   DATA[1411,38] := 0.000128152;
   DATA[1411,39] := 1.0;
   DATA[1412,1] := 812.7283;
   DATA[1412,2] := 1.0;
   DATA[1412,3] := 1.0;
   DATA[1412,4] := 262.5609;
   DATA[1412,5] := 8.46501;
   DATA[1412,6] := 318.2517;
   DATA[1412,8] := 1.0;
   DATA[1412,9] := 1.0;
   DATA[1412,10] := 1.0;
   DATA[1412,11] := 19.69076;
   DATA[1412,12] := 2.216699;
   DATA[1412,13] := 979.9971;
   DATA[1412,14] := 1.0;
   DATA[1412,15] := 2.0;
   DATA[1412,16] := 1.0;
   DATA[1412,17] := 1.0;
   DATA[1412,18] := 1.0;
   DATA[1412,19] := 2.0;
   DATA[1412,20] := 148.808;
   DATA[1412,21] := 153.5247;
   DATA[1412,22] := 1.7057;
   DATA[1412,23] := 779.3771;
   DATA[1412,24] := 2.0;
   DATA[1412,25] := 2.0;
   DATA[1412,26] := 7.877019;
   DATA[1412,27] := 142.707;
   DATA[1412,28] := 263.1056;
   DATA[1412,29] := 12.11228;
   DATA[1412,30] := 1.718662;
   DATA[1412,31] := 1.271679;
   DATA[1412,32] := 0.7352687;
   DATA[1412,33] := 0.3083624;
   DATA[1412,34] := 2.0;
   DATA[1412,35] := 249.5834;
   DATA[1412,36] := 1.569859;
   DATA[1412,37] := 188.4933;
   DATA[1412,38] := 0.000128152;
   DATA[1412,39] := 1.0;
   DATA[1413,1] := 813.1209;
   DATA[1413,2] := 1.0;
   DATA[1413,3] := 1.0;
   DATA[1413,4] := 262.5609;
   DATA[1413,5] := 8.46501;
   DATA[1413,6] := 318.2517;
   DATA[1413,8] := 1.0;
   DATA[1413,9] := 1.0;
   DATA[1413,10] := 1.0;
   DATA[1413,11] := 19.69076;
   DATA[1413,12] := 2.218621;
   DATA[1413,13] := 979.6367;
   DATA[1413,14] := 1.0;
   DATA[1413,15] := 2.0;
   DATA[1413,16] := 1.0;
   DATA[1413,17] := 1.0;
   DATA[1413,18] := 1.0;
   DATA[1413,19] := 2.0;
   DATA[1413,20] := 148.808;
   DATA[1413,21] := 153.5247;
   DATA[1413,22] := 1.709672;
   DATA[1413,23] := 779.6462;
   DATA[1413,24] := 2.0;
   DATA[1413,25] := 2.0;
   DATA[1413,26] := 7.874776;
   DATA[1413,27] := 142.707;
   DATA[1413,28] := 263.1056;
   DATA[1413,29] := 12.11228;
   DATA[1413,30] := 1.720328;
   DATA[1413,31] := 1.277315;
   DATA[1413,32] := 0.7352687;
   DATA[1413,33] := 0.3083624;
   DATA[1413,34] := 2.0;
   DATA[1413,35] := 249.5834;
   DATA[1413,36] := 1.617916;
   DATA[1413,37] := 188.4933;
   DATA[1413,38] := 0.000128152;
   DATA[1413,39] := 1.0;
   DATA[1414,1] := 812.6498;
   DATA[1414,2] := 1.0;
   DATA[1414,3] := 1.0;
   DATA[1414,4] := 262.5609;
   DATA[1414,5] := 8.46501;
   DATA[1414,6] := 318.2517;
   DATA[1414,8] := 1.0;
   DATA[1414,9] := 1.0;
   DATA[1414,10] := 1.0;
   DATA[1414,11] := 19.69076;
   DATA[1414,12] := 2.218621;
   DATA[1414,13] := 978.9557;
   DATA[1414,14] := 1.0;
   DATA[1414,15] := 2.0;
   DATA[1414,16] := 1.0;
   DATA[1414,17] := 1.0;
   DATA[1414,18] := 1.0;
   DATA[1414,19] := 2.0;
   DATA[1414,20] := 148.808;
   DATA[1414,21] := 153.5247;
   DATA[1414,22] := 1.710057;
   DATA[1414,23] := 779.6847;
   DATA[1414,24] := 2.0;
   DATA[1414,25] := 2.0;
   DATA[1414,26] := 7.874776;
   DATA[1414,27] := 142.707;
   DATA[1414,28] := 263.1056;
   DATA[1414,29] := 12.11228;
   DATA[1414,30] := 1.721097;
   DATA[1414,31] := 1.272064;
   DATA[1414,32] := 0.7352687;
   DATA[1414,33] := 0.3083624;
   DATA[1414,34] := 2.0;
   DATA[1414,35] := 249.5834;
   DATA[1414,36] := 1.617916;
   DATA[1414,37] := 188.4933;
   DATA[1414,38] := 0.000128152;
   DATA[1414,39] := 1.0;
   DATA[1415,1] := 812.5714;
   DATA[1415,2] := 1.0;
   DATA[1415,3] := 1.0;
   DATA[1415,4] := 262.5609;
   DATA[1415,5] := 8.46501;
   DATA[1415,6] := 318.2517;
   DATA[1415,8] := 1.0;
   DATA[1415,9] := 1.0;
   DATA[1415,10] := 1.0;
   DATA[1415,11] := 19.7996;
   DATA[1415,12] := 2.218621;
   DATA[1415,13] := 978.5552;
   DATA[1415,14] := 1.0;
   DATA[1415,15] := 2.0;
   DATA[1415,16] := 1.0;
   DATA[1415,17] := 1.0;
   DATA[1415,18] := 1.0;
   DATA[1415,19] := 2.0;
   DATA[1415,20] := 148.808;
   DATA[1415,21] := 153.5247;
   DATA[1415,22] := 1.710954;
   DATA[1415,23] := 780.0308;
   DATA[1415,24] := 2.0;
   DATA[1415,25] := 2.0;
   DATA[1415,26] := 7.874776;
   DATA[1415,27] := 142.707;
   DATA[1415,28] := 263.1056;
   DATA[1415,29] := 12.11228;
   DATA[1415,30] := 1.722251;
   DATA[1415,31] := 1.271295;
   DATA[1415,32] := 0.7352687;
   DATA[1415,33] := 0.3083624;
   DATA[1415,34] := 2.0;
   DATA[1415,35] := 249.5834;
   DATA[1415,36] := 1.617916;
   DATA[1415,37] := 188.4933;
   DATA[1415,38] := 0.000128152;
   DATA[1415,39] := 1.0;
   DATA[1416,1] := 812.8461;
   DATA[1416,2] := 1.0;
   DATA[1416,3] := 1.0;
   DATA[1416,4] := 262.5609;
   DATA[1416,5] := 8.46501;
   DATA[1416,6] := 318.2517;
   DATA[1416,8] := 1.0;
   DATA[1416,9] := 1.0;
   DATA[1416,10] := 1.0;
   DATA[1416,11] := 19.81881;
   DATA[1416,12] := 2.218621;
   DATA[1416,13] := 978.4351;
   DATA[1416,14] := 1.0;
   DATA[1416,15] := 2.0;
   DATA[1416,16] := 1.0;
   DATA[1416,17] := 1.0;
   DATA[1416,18] := 1.0;
   DATA[1416,19] := 2.0;
   DATA[1416,20] := 148.808;
   DATA[1416,21] := 153.5247;
   DATA[1416,22] := 1.710954;
   DATA[1416,23] := 780.1461;
   DATA[1416,24] := 2.0;
   DATA[1416,25] := 2.0;
   DATA[1416,26] := 7.874776;
   DATA[1416,27] := 142.707;
   DATA[1416,28] := 263.1056;
   DATA[1416,29] := 12.11228;
   DATA[1416,30] := 1.722251;
   DATA[1416,31] := 1.271295;
   DATA[1416,32] := 0.7352687;
   DATA[1416,33] := 0.3083624;
   DATA[1416,34] := 2.0;
   DATA[1416,35] := 249.5834;
   DATA[1416,36] := 1.617916;
   DATA[1416,37] := 188.4933;
   DATA[1416,38] := 0.000128152;
   DATA[1416,39] := 1.0;
   DATA[1417,1] := 812.9246;
   DATA[1417,2] := 1.0;
   DATA[1417,3] := 1.0;
   DATA[1417,4] := 262.5609;
   DATA[1417,5] := 8.46501;
   DATA[1417,6] := 318.2517;
   DATA[1417,8] := 1.0;
   DATA[1417,9] := 1.0;
   DATA[1417,10] := 1.0;
   DATA[1417,11] := 19.81881;
   DATA[1417,12] := 2.218621;
   DATA[1417,13] := 978.0345;
   DATA[1417,14] := 1.0;
   DATA[1417,15] := 2.0;
   DATA[1417,16] := 1.0;
   DATA[1417,17] := 1.0;
   DATA[1417,18] := 1.0;
   DATA[1417,19] := 2.0;
   DATA[1417,20] := 148.808;
   DATA[1417,21] := 153.5247;
   DATA[1417,22] := 1.710954;
   DATA[1417,23] := 780.4537;
   DATA[1417,24] := 2.0;
   DATA[1417,25] := 2.0;
   DATA[1417,26] := 7.874776;
   DATA[1417,27] := 142.707;
   DATA[1417,28] := 263.1056;
   DATA[1417,29] := 12.11228;
   DATA[1417,30] := 1.722251;
   DATA[1417,31] := 1.271295;
   DATA[1417,32] := 0.7352687;
   DATA[1417,33] := 0.3083624;
   DATA[1417,34] := 2.0;
   DATA[1417,35] := 249.5834;
   DATA[1417,36] := 1.617916;
   DATA[1417,37] := 188.4933;
   DATA[1417,38] := 0.000128152;
   DATA[1417,39] := 1.0;
   DATA[1418,1] := 813.0031;
   DATA[1418,2] := 1.0;
   DATA[1418,3] := 1.0;
   DATA[1418,4] := 262.5609;
   DATA[1418,5] := 8.46501;
   DATA[1418,6] := 318.2517;
   DATA[1418,8] := 1.0;
   DATA[1418,9] := 1.0;
   DATA[1418,10] := 1.0;
   DATA[1418,11] := 19.76759;
   DATA[1418,12] := 2.218621;
   DATA[1418,13] := 977.7942;
   DATA[1418,14] := 1.0;
   DATA[1418,15] := 2.0;
   DATA[1418,16] := 1.0;
   DATA[1418,17] := 1.0;
   DATA[1418,18] := 1.0;
   DATA[1418,19] := 2.0;
   DATA[1418,20] := 148.808;
   DATA[1418,21] := 153.5247;
   DATA[1418,22] := 1.710954;
   DATA[1418,23] := 780.7229;
   DATA[1418,24] := 2.0;
   DATA[1418,25] := 2.0;
   DATA[1418,26] := 7.874776;
   DATA[1418,27] := 142.707;
   DATA[1418,28] := 263.1056;
   DATA[1418,29] := 12.11228;
   DATA[1418,30] := 1.722251;
   DATA[1418,31] := 1.262969;
   DATA[1418,32] := 0.7352687;
   DATA[1418,33] := 0.3083624;
   DATA[1418,34] := 2.0;
   DATA[1418,35] := 249.5834;
   DATA[1418,36] := 1.617916;
   DATA[1418,37] := 188.4933;
   DATA[1418,38] := 0.000128152;
   DATA[1418,39] := 1.0;
   DATA[1419,1] := 813.3564;
   DATA[1419,2] := 1.0;
   DATA[1419,3] := 1.0;
   DATA[1419,4] := 262.5609;
   DATA[1419,5] := 8.46501;
   DATA[1419,6] := 318.2517;
   DATA[1419,8] := 1.0;
   DATA[1419,9] := 1.0;
   DATA[1419,10] := 1.0;
   DATA[1419,11] := 19.76759;
   DATA[1419,12] := 2.218621;
   DATA[1419,13] := 977.1533;
   DATA[1419,14] := 1.0;
   DATA[1419,15] := 2.0;
   DATA[1419,16] := 1.0;
   DATA[1419,17] := 1.0;
   DATA[1419,18] := 1.0;
   DATA[1419,19] := 2.0;
   DATA[1419,20] := 148.808;
   DATA[1419,21] := 153.5247;
   DATA[1419,22] := 1.712363;
   DATA[1419,23] := 781.1459;
   DATA[1419,24] := 2.0;
   DATA[1419,25] := 2.0;
   DATA[1419,26] := 7.87766;
   DATA[1419,27] := 142.707;
   DATA[1419,28] := 263.1056;
   DATA[1419,29] := 12.11228;
   DATA[1419,30] := 1.722251;
   DATA[1419,31] := 1.274881;
   DATA[1419,32] := 0.7352687;
   DATA[1419,33] := 0.3083624;
   DATA[1419,34] := 2.0;
   DATA[1419,35] := 249.5834;
   DATA[1419,36] := 1.617916;
   DATA[1419,37] := 188.4933;
   DATA[1419,38] := 0.000128152;
   DATA[1419,39] := 1.0;
   DATA[1420,1] := 813.5527;
   DATA[1420,2] := 1.0;
   DATA[1420,3] := 1.0;
   DATA[1420,4] := 262.5609;
   DATA[1420,5] := 8.46501;
   DATA[1420,6] := 318.3799;
   DATA[1420,8] := 1.0;
   DATA[1420,9] := 1.0;
   DATA[1420,10] := 1.0;
   DATA[1420,11] := 19.73558;
   DATA[1420,12] := 2.218621;
   DATA[1420,13] := 976.5926;
   DATA[1420,14] := 1.0;
   DATA[1420,15] := 2.0;
   DATA[1420,16] := 1.0;
   DATA[1420,17] := 1.0;
   DATA[1420,18] := 1.0;
   DATA[1420,19] := 2.0;
   DATA[1420,20] := 148.808;
   DATA[1420,21] := 153.5247;
   DATA[1420,22] := 1.712363;
   DATA[1420,23] := 780.9536;
   DATA[1420,24] := 2.0;
   DATA[1420,25] := 2.0;
   DATA[1420,26] := 7.87766;
   DATA[1420,27] := 142.707;
   DATA[1420,28] := 263.1056;
   DATA[1420,29] := 12.11228;
   DATA[1420,30] := 1.722251;
   DATA[1420,31] := 1.288203;
   DATA[1420,32] := 0.7352687;
   DATA[1420,33] := 0.3083624;
   DATA[1420,34] := 2.0;
   DATA[1420,35] := 249.5834;
   DATA[1420,36] := 1.617916;
   DATA[1420,37] := 188.4933;
   DATA[1420,38] := 0.000128152;
   DATA[1420,39] := 1.0;
   DATA[1421,1] := 813.7097;
   DATA[1421,2] := 1.0;
   DATA[1421,3] := 1.0;
   DATA[1421,4] := 262.5609;
   DATA[1421,5] := 8.46501;
   DATA[1421,6] := 318.3799;
   DATA[1421,8] := 1.0;
   DATA[1421,9] := 1.0;
   DATA[1421,10] := 1.0;
   DATA[1421,11] := 19.7804;
   DATA[1421,12] := 2.218621;
   DATA[1421,13] := 976.192;
   DATA[1421,14] := 1.0;
   DATA[1421,15] := 2.0;
   DATA[1421,16] := 1.0;
   DATA[1421,17] := 1.0;
   DATA[1421,18] := 1.0;
   DATA[1421,19] := 2.0;
   DATA[1421,20] := 148.808;
   DATA[1421,21] := 153.5247;
   DATA[1421,22] := 1.712363;
   DATA[1421,23] := 781.2228;
   DATA[1421,24] := 2.0;
   DATA[1421,25] := 2.0;
   DATA[1421,26] := 7.87766;
   DATA[1421,27] := 142.707;
   DATA[1421,28] := 263.1056;
   DATA[1421,29] := 12.11228;
   DATA[1421,30] := 1.722251;
   DATA[1421,31] := 1.29781;
   DATA[1421,32] := 0.7352687;
   DATA[1421,33] := 0.3083624;
   DATA[1421,34] := 2.0;
   DATA[1421,35] := 249.7597;
   DATA[1421,36] := 1.617916;
   DATA[1421,37] := 188.7016;
   DATA[1421,38] := 0.000128152;
   DATA[1421,39] := 1.0;
   DATA[1422,1] := 813.5134;
   DATA[1422,2] := 1.0;
   DATA[1422,3] := 1.0;
   DATA[1422,4] := 262.5609;
   DATA[1422,5] := 8.46501;
   DATA[1422,6] := 318.3799;
   DATA[1422,8] := 1.0;
   DATA[1422,9] := 1.0;
   DATA[1422,10] := 1.0;
   DATA[1422,11] := 19.7804;
   DATA[1422,12] := 2.218621;
   DATA[1422,13] := 975.5511;
   DATA[1422,14] := 1.0;
   DATA[1422,15] := 2.0;
   DATA[1422,16] := 1.0;
   DATA[1422,17] := 1.0;
   DATA[1422,18] := 1.0;
   DATA[1422,19] := 2.0;
   DATA[1422,20] := 148.808;
   DATA[1422,21] := 153.5247;
   DATA[1422,22] := 1.710698;
   DATA[1422,23] := 781.415;
   DATA[1422,24] := 2.0;
   DATA[1422,25] := 2.0;
   DATA[1422,26] := 7.87766;
   DATA[1422,27] := 142.707;
   DATA[1422,28] := 263.1056;
   DATA[1422,29] := 12.11228;
   DATA[1422,30] := 1.722251;
   DATA[1422,31] := 1.30921;
   DATA[1422,32] := 0.7352687;
   DATA[1422,33] := 0.3083624;
   DATA[1422,34] := 2.0;
   DATA[1422,35] := 249.8398;
   DATA[1422,36] := 1.617916;
   DATA[1422,37] := 188.7657;
   DATA[1422,38] := 0.000128152;
   DATA[1422,39] := 1.0;
   DATA[1423,1] := 813.6312;
   DATA[1423,2] := 1.0;
   DATA[1423,3] := 1.0;
   DATA[1423,4] := 262.5609;
   DATA[1423,5] := 8.46501;
   DATA[1423,6] := 318.3799;
   DATA[1423,8] := 1.0;
   DATA[1423,9] := 1.0;
   DATA[1423,10] := 1.0;
   DATA[1423,11] := 19.7804;
   DATA[1423,12] := 2.216699;
   DATA[1423,13] := 975.0305;
   DATA[1423,14] := 1.0;
   DATA[1423,15] := 2.0;
   DATA[1423,16] := 1.0;
   DATA[1423,17] := 1.0;
   DATA[1423,18] := 1.0;
   DATA[1423,19] := 2.0;
   DATA[1423,20] := 148.808;
   DATA[1423,21] := 153.5247;
   DATA[1423,22] := 1.7098;
   DATA[1423,23] := 781.3381;
   DATA[1423,24] := 2.0;
   DATA[1423,25] := 2.0;
   DATA[1423,26] := 7.87766;
   DATA[1423,27] := 142.707;
   DATA[1423,28] := 263.1056;
   DATA[1423,29] := 12.11228;
   DATA[1423,30] := 1.722251;
   DATA[1423,31] := 1.311643;
   DATA[1423,32] := 0.7359089;
   DATA[1423,33] := 0.3083624;
   DATA[1423,34] := 2.0;
   DATA[1423,35] := 249.8398;
   DATA[1423,36] := 1.617916;
   DATA[1423,37] := 188.7657;
   DATA[1423,38] := 0.000128152;
   DATA[1423,39] := 1.0;
   DATA[1424,1] := 813.7097;
   DATA[1424,2] := 1.0;
   DATA[1424,3] := 1.0;
   DATA[1424,4] := 262.5609;
   DATA[1424,5] := 8.46501;
   DATA[1424,6] := 318.3799;
   DATA[1424,8] := 1.0;
   DATA[1424,9] := 1.0;
   DATA[1424,10] := 1.0;
   DATA[1424,11] := 19.67796;
   DATA[1424,12] := 2.216699;
   DATA[1424,13] := 974.7902;
   DATA[1424,14] := 1.0;
   DATA[1424,15] := 2.0;
   DATA[1424,16] := 1.0;
   DATA[1424,17] := 1.0;
   DATA[1424,18] := 1.0;
   DATA[1424,19] := 2.0;
   DATA[1424,20] := 148.808;
   DATA[1424,21] := 153.5247;
   DATA[1424,22] := 1.7098;
   DATA[1424,23] := 781.5304;
   DATA[1424,24] := 2.0;
   DATA[1424,25] := 2.0;
   DATA[1424,26] := 7.87766;
   DATA[1424,27] := 142.707;
   DATA[1424,28] := 263.1056;
   DATA[1424,29] := 12.11228;
   DATA[1424,30] := 1.720841;
   DATA[1424,31] := 1.302037;
   DATA[1424,32] := 0.736549;
   DATA[1424,33] := 0.3083624;
   DATA[1424,34] := 2.0;
   DATA[1424,35] := 249.8398;
   DATA[1424,36] := 1.617916;
   DATA[1424,37] := 188.7657;
   DATA[1424,38] := 0.000128152;
   DATA[1424,39] := 1.0;
   DATA[1425,1] := 813.6312;
   DATA[1425,2] := 1.0;
   DATA[1425,3] := 1.0;
   DATA[1425,4] := 262.5609;
   DATA[1425,5] := 8.46501;
   DATA[1425,6] := 318.3799;
   DATA[1425,8] := 1.0;
   DATA[1425,9] := 1.0;
   DATA[1425,10] := 1.0;
   DATA[1425,11] := 19.67796;
   DATA[1425,12] := 2.218621;
   DATA[1425,13] := 974.6299;
   DATA[1425,14] := 1.0;
   DATA[1425,15] := 2.0;
   DATA[1425,16] := 1.0;
   DATA[1425,17] := 1.0;
   DATA[1425,18] := 1.0;
   DATA[1425,19] := 2.0;
   DATA[1425,20] := 148.808;
   DATA[1425,21] := 153.5247;
   DATA[1425,22] := 1.7098;
   DATA[1425,23] := 781.6073;
   DATA[1425,24] := 2.0;
   DATA[1425,25] := 2.0;
   DATA[1425,26] := 7.87766;
   DATA[1425,27] := 142.707;
   DATA[1425,28] := 263.1056;
   DATA[1425,29] := 12.11228;
   DATA[1425,30] := 1.718662;
   DATA[1425,31] := 1.302037;
   DATA[1425,32] := 0.736549;
   DATA[1425,33] := 0.3083624;
   DATA[1425,34] := 2.0;
   DATA[1425,35] := 249.8398;
   DATA[1425,36] := 1.617916;
   DATA[1425,37] := 188.7657;
   DATA[1425,38] := 0.000128152;
   DATA[1425,39] := 1.0;
   DATA[1426,1] := 813.1994;
   DATA[1426,2] := 1.0;
   DATA[1426,3] := 1.0;
   DATA[1426,4] := 262.5609;
   DATA[1426,5] := 8.46501;
   DATA[1426,6] := 318.3799;
   DATA[1426,8] := 1.0;
   DATA[1426,9] := 1.0;
   DATA[1426,10] := 1.0;
   DATA[1426,11] := 19.73558;
   DATA[1426,12] := 2.219005;
   DATA[1426,13] := 974.4697;
   DATA[1426,14] := 1.0;
   DATA[1426,15] := 2.0;
   DATA[1426,16] := 1.0;
   DATA[1426,17] := 1.0;
   DATA[1426,18] := 1.0;
   DATA[1426,19] := 2.0;
   DATA[1426,20] := 148.808;
   DATA[1426,21] := 153.5247;
   DATA[1426,22] := 1.7098;
   DATA[1426,23] := 781.9918;
   DATA[1426,24] := 2.0;
   DATA[1426,25] := 2.0;
   DATA[1426,26] := 7.87766;
   DATA[1426,27] := 142.707;
   DATA[1426,28] := 263.1056;
   DATA[1426,29] := 12.11228;
   DATA[1426,30] := 1.718662;
   DATA[1426,31] := 1.295248;
   DATA[1426,32] := 0.7380853;
   DATA[1426,33] := 0.3083624;
   DATA[1426,34] := 2.0;
   DATA[1426,35] := 249.8398;
   DATA[1426,36] := 1.617916;
   DATA[1426,37] := 188.7657;
   DATA[1426,38] := 0.000128152;
   DATA[1426,39] := 1.0;
   DATA[1427,1] := 813.1994;
   DATA[1427,2] := 1.0;
   DATA[1427,3] := 1.0;
   DATA[1427,4] := 262.5609;
   DATA[1427,5] := 8.46501;
   DATA[1427,6] := 318.3799;
   DATA[1427,8] := 1.0;
   DATA[1427,9] := 1.0;
   DATA[1427,10] := 1.0;
   DATA[1427,11] := 19.79;
   DATA[1427,12] := 2.219005;
   DATA[1427,13] := 973.9891;
   DATA[1427,14] := 1.0;
   DATA[1427,15] := 2.0;
   DATA[1427,16] := 1.0;
   DATA[1427,17] := 1.0;
   DATA[1427,18] := 1.0;
   DATA[1427,19] := 2.0;
   DATA[1427,20] := 148.808;
   DATA[1427,21] := 153.5247;
   DATA[1427,22] := 1.7098;
   DATA[1427,23] := 781.7227;
   DATA[1427,24] := 2.0;
   DATA[1427,25] := 2.0;
   DATA[1427,26] := 7.87766;
   DATA[1427,27] := 142.707;
   DATA[1427,28] := 263.1056;
   DATA[1427,29] := 12.11228;
   DATA[1427,30] := 1.718662;
   DATA[1427,31] := 1.282439;
   DATA[1427,32] := 0.7387255;
   DATA[1427,33] := 0.3083624;
   DATA[1427,34] := 2.0;
   DATA[1427,35] := 249.8398;
   DATA[1427,36] := 1.617916;
   DATA[1427,37] := 188.6375;
   DATA[1427,38] := 0.000128152;
   DATA[1427,39] := 1.0;
   DATA[1428,1] := 813.4349;
   DATA[1428,2] := 1.0;
   DATA[1428,3] := 1.0;
   DATA[1428,4] := 262.5609;
   DATA[1428,5] := 8.46501;
   DATA[1428,6] := 318.3799;
   DATA[1428,8] := 1.0;
   DATA[1428,9] := 1.0;
   DATA[1428,10] := 1.0;
   DATA[1428,11] := 19.79;
   DATA[1428,12] := 2.217211;
   DATA[1428,13] := 973.1479;
   DATA[1428,14] := 1.0;
   DATA[1428,15] := 2.0;
   DATA[1428,16] := 1.0;
   DATA[1428,17] := 1.0;
   DATA[1428,18] := 1.0;
   DATA[1428,19] := 2.0;
   DATA[1428,20] := 148.808;
   DATA[1428,21] := 153.5247;
   DATA[1428,22] := 1.7098;
   DATA[1428,23] := 781.8765;
   DATA[1428,24] := 2.0;
   DATA[1428,25] := 2.0;
   DATA[1428,26] := 7.877339;
   DATA[1428,27] := 142.707;
   DATA[1428,28] := 263.1056;
   DATA[1428,29] := 12.11228;
   DATA[1428,30] := 1.718662;
   DATA[1428,31] := 1.272576;
   DATA[1428,32] := 0.7387255;
   DATA[1428,33] := 0.3083624;
   DATA[1428,34] := 2.0;
   DATA[1428,35] := 249.8398;
   DATA[1428,36] := 1.617916;
   DATA[1428,37] := 188.6215;
   DATA[1428,38] := 0.000128152;
   DATA[1428,39] := 1.0;
   DATA[1429,1] := 813.5527;
   DATA[1429,2] := 1.0;
   DATA[1429,3] := 1.0;
   DATA[1429,4] := 262.5609;
   DATA[1429,5] := 8.466932;
   DATA[1429,6] := 318.3799;
   DATA[1429,8] := 1.0;
   DATA[1429,9] := 1.0;
   DATA[1429,10] := 1.0;
   DATA[1429,11] := 19.7804;
   DATA[1429,12] := 2.217211;
   DATA[1429,13] := 972.3869;
   DATA[1429,14] := 1.0;
   DATA[1429,15] := 2.0;
   DATA[1429,16] := 1.0;
   DATA[1429,17] := 1.0;
   DATA[1429,18] := 1.0;
   DATA[1429,19] := 2.0;
   DATA[1429,20] := 148.808;
   DATA[1429,21] := 153.5247;
   DATA[1429,22] := 1.7098;
   DATA[1429,23] := 782.261;
   DATA[1429,24] := 2.0;
   DATA[1429,25] := 2.0;
   DATA[1429,26] := 7.877339;
   DATA[1429,27] := 142.707;
   DATA[1429,28] := 263.1056;
   DATA[1429,29] := 12.11228;
   DATA[1429,30] := 1.718662;
   DATA[1429,31] := 1.262073;
   DATA[1429,32] := 0.7387255;
   DATA[1429,33] := 0.3083624;
   DATA[1429,34] := 2.0;
   DATA[1429,35] := 249.6635;
   DATA[1429,36] := 1.617916;
   DATA[1429,37] := 188.6215;
   DATA[1429,38] := 0.000128152;
   DATA[1429,39] := 1.0;
   DATA[1430,1] := 813.5919;
   DATA[1430,2] := 1.0;
   DATA[1430,3] := 1.0;
   DATA[1430,4] := 262.5609;
   DATA[1430,5] := 8.468855;
   DATA[1430,6] := 318.3799;
   DATA[1430,8] := 1.0;
   DATA[1430,9] := 1.0;
   DATA[1430,10] := 1.0;
   DATA[1430,11] := 19.7804;
   DATA[1430,12] := 2.216827;
   DATA[1430,13] := 972.1466;
   DATA[1430,14] := 1.0;
   DATA[1430,15] := 2.0;
   DATA[1430,16] := 1.0;
   DATA[1430,17] := 1.0;
   DATA[1430,18] := 1.0;
   DATA[1430,19] := 2.0;
   DATA[1430,20] := 148.808;
   DATA[1430,21] := 153.5247;
   DATA[1430,22] := 1.7098;
   DATA[1430,23] := 782.2994;
   DATA[1430,24] := 2.0;
   DATA[1430,25] := 2.0;
   DATA[1430,26] := 7.877339;
   DATA[1430,27] := 142.707;
   DATA[1430,28] := 263.1056;
   DATA[1430,29] := 12.11228;
   DATA[1430,30] := 1.718662;
   DATA[1430,31] := 1.262073;
   DATA[1430,32] := 0.7370611;
   DATA[1430,33] := 0.3083624;
   DATA[1430,34] := 2.0;
   DATA[1430,35] := 249.6635;
   DATA[1430,36] := 1.617916;
   DATA[1430,37] := 188.6215;
   DATA[1430,38] := 0.000128152;
   DATA[1430,39] := 1.0;
   DATA[1431,1] := 813.7489;
   DATA[1431,2] := 1.0;
   DATA[1431,3] := 1.0;
   DATA[1431,4] := 262.5609;
   DATA[1431,5] := 8.468855;
   DATA[1431,6] := 318.3799;
   DATA[1431,8] := 1.0;
   DATA[1431,9] := 1.0;
   DATA[1431,10] := 1.0;
   DATA[1431,11] := 19.7804;
   DATA[1431,12] := 2.216827;
   DATA[1431,13] := 971.5858;
   DATA[1431,14] := 1.0;
   DATA[1431,15] := 2.0;
   DATA[1431,16] := 1.0;
   DATA[1431,17] := 1.0;
   DATA[1431,18] := 1.0;
   DATA[1431,19] := 2.0;
   DATA[1431,20] := 148.808;
   DATA[1431,21] := 153.5247;
   DATA[1431,22] := 1.711466;
   DATA[1431,23] := 782.2994;
   DATA[1431,24] := 2.0;
   DATA[1431,25] := 2.0;
   DATA[1431,26] := 7.876058;
   DATA[1431,27] := 142.707;
   DATA[1431,28] := 263.1056;
   DATA[1431,29] := 12.11228;
   DATA[1431,30] := 1.719046;
   DATA[1431,31] := 1.280646;
   DATA[1431,32] := 0.7355248;
   DATA[1431,33] := 0.3083624;
   DATA[1431,34] := 2.0;
   DATA[1431,35] := 249.6635;
   DATA[1431,36] := 1.617916;
   DATA[1431,37] := 188.6215;
   DATA[1431,38] := 0.000128152;
   DATA[1431,39] := 1.0;
   DATA[1432,1] := 813.6312;
   DATA[1432,2] := 1.0;
   DATA[1432,3] := 1.0;
   DATA[1432,4] := 262.5609;
   DATA[1432,5] := 8.468855;
   DATA[1432,6] := 318.3799;
   DATA[1432,8] := 1.0;
   DATA[1432,9] := 1.0;
   DATA[1432,10] := 1.0;
   DATA[1432,11] := 19.7804;
   DATA[1432,12] := 2.216827;
   DATA[1432,13] := 971.2253;
   DATA[1432,14] := 1.0;
   DATA[1432,15] := 2.0;
   DATA[1432,16] := 1.0;
   DATA[1432,17] := 1.0;
   DATA[1432,18] := 1.0;
   DATA[1432,19] := 2.0;
   DATA[1432,20] := 148.808;
   DATA[1432,21] := 153.5247;
   DATA[1432,22] := 1.711466;
   DATA[1432,23] := 782.261;
   DATA[1432,24] := 2.0;
   DATA[1432,25] := 2.0;
   DATA[1432,26] := 7.875737;
   DATA[1432,27] := 142.707;
   DATA[1432,28] := 263.1056;
   DATA[1432,29] := 12.11228;
   DATA[1432,30] := 1.719559;
   DATA[1432,31] := 1.292558;
   DATA[1432,32] := 0.7352687;
   DATA[1432,33] := 0.3083624;
   DATA[1432,34] := 2.0;
   DATA[1432,35] := 249.6635;
   DATA[1432,36] := 1.617916;
   DATA[1432,37] := 188.6215;
   DATA[1432,38] := 0.000128152;
   DATA[1432,39] := 1.0;
   DATA[1433,1] := 813.9452;
   DATA[1433,2] := 1.0;
   DATA[1433,3] := 1.0;
   DATA[1433,4] := 262.5609;
   DATA[1433,5] := 8.468855;
   DATA[1433,6] := 318.3799;
   DATA[1433,8] := 1.0;
   DATA[1433,9] := 1.0;
   DATA[1433,10] := 1.0;
   DATA[1433,11] := 19.76439;
   DATA[1433,12] := 2.218621;
   DATA[1433,13] := 971.0651;
   DATA[1433,14] := 1.0;
   DATA[1433,15] := 2.0;
   DATA[1433,16] := 1.0;
   DATA[1433,17] := 1.0;
   DATA[1433,18] := 1.0;
   DATA[1433,19] := 2.0;
   DATA[1433,20] := 148.808;
   DATA[1433,21] := 153.5247;
   DATA[1433,22] := 1.711466;
   DATA[1433,23] := 782.4532;
   DATA[1433,24] := 2.0;
   DATA[1433,25] := 2.0;
   DATA[1433,26] := 7.875737;
   DATA[1433,27] := 142.707;
   DATA[1433,28] := 263.1056;
   DATA[1433,29] := 12.11228;
   DATA[1433,30] := 1.72161;
   DATA[1433,31] := 1.292558;
   DATA[1433,32] := 0.7352687;
   DATA[1433,33] := 0.3083624;
   DATA[1433,34] := 2.0;
   DATA[1433,35] := 249.6635;
   DATA[1433,36] := 1.617916;
   DATA[1433,37] := 188.6215;
   DATA[1433,38] := 0.000128152;
   DATA[1433,39] := 1.0;
   DATA[1434,1] := 813.7882;
   DATA[1434,2] := 1.0;
   DATA[1434,3] := 1.0;
   DATA[1434,4] := 262.5609;
   DATA[1434,5] := 8.468855;
   DATA[1434,6] := 318.3799;
   DATA[1434,8] := 1.0;
   DATA[1434,9] := 1.0;
   DATA[1434,10] := 1.0;
   DATA[1434,11] := 19.76439;
   DATA[1434,12] := 2.218621;
   DATA[1434,13] := 970.6245;
   DATA[1434,14] := 1.0;
   DATA[1434,15] := 2.0;
   DATA[1434,16] := 1.0;
   DATA[1434,17] := 1.0;
   DATA[1434,18] := 1.0;
   DATA[1434,19] := 2.0;
   DATA[1434,20] := 148.808;
   DATA[1434,21] := 153.5247;
   DATA[1434,22] := 1.711466;
   DATA[1434,23] := 782.4532;
   DATA[1434,24] := 2.0;
   DATA[1434,25] := 2.0;
   DATA[1434,26] := 7.875737;
   DATA[1434,27] := 142.707;
   DATA[1434,28] := 263.1056;
   DATA[1434,29] := 12.11228;
   DATA[1434,30] := 1.722379;
   DATA[1434,31] := 1.289996;
   DATA[1434,32] := 0.7352687;
   DATA[1434,33] := 0.3083624;
   DATA[1434,34] := 2.0;
   DATA[1434,35] := 249.8558;
   DATA[1434,36] := 1.617916;
   DATA[1434,37] := 188.6215;
   DATA[1434,38] := 0.000128152;
   DATA[1434,39] := 1.0;
   DATA[1435,1] := 813.5134;
   DATA[1435,2] := 1.0;
   DATA[1435,3] := 1.0;
   DATA[1435,4] := 262.5609;
   DATA[1435,5] := 8.466612;
   DATA[1435,6] := 318.3799;
   DATA[1435,8] := 1.0;
   DATA[1435,9] := 1.0;
   DATA[1435,10] := 1.0;
   DATA[1435,11] := 19.84442;
   DATA[1435,12] := 2.217468;
   DATA[1435,13] := 970.264;
   DATA[1435,14] := 1.0;
   DATA[1435,15] := 2.0;
   DATA[1435,16] := 1.0;
   DATA[1435,17] := 1.0;
   DATA[1435,18] := 1.0;
   DATA[1435,19] := 2.0;
   DATA[1435,20] := 148.808;
   DATA[1435,21] := 153.5247;
   DATA[1435,22] := 1.711466;
   DATA[1435,23] := 782.607;
   DATA[1435,24] := 2.0;
   DATA[1435,25] := 2.0;
   DATA[1435,26] := 7.875737;
   DATA[1435,27] := 142.707;
   DATA[1435,28] := 263.0095;
   DATA[1435,29] := 12.11228;
   DATA[1435,30] := 1.722379;
   DATA[1435,31] := 1.281927;
   DATA[1435,32] := 0.7352687;
   DATA[1435,33] := 0.3083624;
   DATA[1435,34] := 2.0;
   DATA[1435,35] := 250.0;
   DATA[1435,36] := 1.617916;
   DATA[1435,37] := 188.8779;
   DATA[1435,38] := 0.000128152;
   DATA[1435,39] := 1.0;
   DATA[1436,1] := 813.3171;
   DATA[1436,2] := 1.0;
   DATA[1436,3] := 1.0;
   DATA[1436,4] := 262.5609;
   DATA[1436,5] := 8.464369;
   DATA[1436,6] := 318.3799;
   DATA[1436,8] := 1.0;
   DATA[1436,9] := 1.0;
   DATA[1436,10] := 1.0;
   DATA[1436,11] := 19.88604;
   DATA[1436,12] := 2.216571;
   DATA[1436,13] := 970.0237;
   DATA[1436,14] := 1.0;
   DATA[1436,15] := 2.0;
   DATA[1436,16] := 1.0;
   DATA[1436,17] := 1.0;
   DATA[1436,18] := 1.0;
   DATA[1436,19] := 2.0;
   DATA[1436,20] := 148.808;
   DATA[1436,21] := 153.5247;
   DATA[1436,22] := 1.711466;
   DATA[1436,23] := 782.7608;
   DATA[1436,24] := 2.0;
   DATA[1436,25] := 2.0;
   DATA[1436,26] := 7.875737;
   DATA[1436,27] := 142.707;
   DATA[1436,28] := 263.0095;
   DATA[1436,29] := 12.11228;
   DATA[1436,30] := 1.722379;
   DATA[1436,31] := 1.281542;
   DATA[1436,32] := 0.7352687;
   DATA[1436,33] := 0.3083624;
   DATA[1436,34] := 2.0;
   DATA[1436,35] := 250.0961;
   DATA[1436,36] := 1.617916;
   DATA[1436,37] := 188.974;
   DATA[1436,38] := 0.000128152;
   DATA[1436,39] := 1.0;
   DATA[1437,1] := 813.1994;
   DATA[1437,2] := 1.0;
   DATA[1437,3] := 1.0;
   DATA[1437,4] := 262.5609;
   DATA[1437,5] := 8.464369;
   DATA[1437,6] := 318.3799;
   DATA[1437,8] := 1.0;
   DATA[1437,9] := 1.0;
   DATA[1437,10] := 1.0;
   DATA[1437,11] := 19.88604;
   DATA[1437,12] := 2.217211;
   DATA[1437,13] := 969.3829;
   DATA[1437,14] := 1.0;
   DATA[1437,15] := 2.0;
   DATA[1437,16] := 1.0;
   DATA[1437,17] := 1.0;
   DATA[1437,18] := 1.0;
   DATA[1437,19] := 2.0;
   DATA[1437,20] := 148.808;
   DATA[1437,21] := 153.5247;
   DATA[1437,22] := 1.711466;
   DATA[1437,23] := 782.9531;
   DATA[1437,24] := 2.0;
   DATA[1437,25] := 2.0;
   DATA[1437,26] := 7.875737;
   DATA[1437,27] := 142.707;
   DATA[1437,28] := 263.0095;
   DATA[1437,29] := 12.11228;
   DATA[1437,30] := 1.72443;
   DATA[1437,31] := 1.282439;
   DATA[1437,32] := 0.7352687;
   DATA[1437,33] := 0.3083624;
   DATA[1437,34] := 2.0;
   DATA[1437,35] := 250.2243;
   DATA[1437,36] := 1.649953;
   DATA[1437,37] := 188.974;
   DATA[1437,38] := 0.000128152;
   DATA[1437,39] := 1.0;
   DATA[1438,1] := 813.2386;
   DATA[1438,2] := 1.0;
   DATA[1438,3] := 1.0;
   DATA[1438,4] := 262.5609;
   DATA[1438,5] := 8.464369;
   DATA[1438,6] := 318.3799;
   DATA[1438,8] := 1.0;
   DATA[1438,9] := 1.0;
   DATA[1438,10] := 1.0;
   DATA[1438,11] := 19.7996;
   DATA[1438,12] := 2.217211;
   DATA[1438,13] := 968.8622;
   DATA[1438,14] := 1.0;
   DATA[1438,15] := 2.0;
   DATA[1438,16] := 1.0;
   DATA[1438,17] := 1.0;
   DATA[1438,18] := 1.0;
   DATA[1438,19] := 2.0;
   DATA[1438,20] := 148.808;
   DATA[1438,21] := 153.5247;
   DATA[1438,22] := 1.711466;
   DATA[1438,23] := 783.03;
   DATA[1438,24] := 2.0;
   DATA[1438,25] := 2.0;
   DATA[1438,26] := 7.875737;
   DATA[1438,27] := 142.707;
   DATA[1438,28] := 263.0095;
   DATA[1438,29] := 12.11228;
   DATA[1438,30] := 1.725968;
   DATA[1438,31] := 1.300115;
   DATA[1438,32] := 0.7352687;
   DATA[1438,33] := 0.3083624;
   DATA[1438,34] := 2.0;
   DATA[1438,35] := 250.2243;
   DATA[1438,36] := 1.649953;
   DATA[1438,37] := 189.1022;
   DATA[1438,38] := 0.000128152;
   DATA[1438,39] := 1.0;
   DATA[1439,1] := 813.0424;
   DATA[1439,2] := 1.0;
   DATA[1439,3] := 1.0;
   DATA[1439,4] := 262.5609;
   DATA[1439,5] := 8.464369;
   DATA[1439,6] := 318.3799;
   DATA[1439,8] := 1.0;
   DATA[1439,9] := 1.0;
   DATA[1439,10] := 1.0;
   DATA[1439,11] := 19.73558;
   DATA[1439,12] := 2.217211;
   DATA[1439,13] := 968.3415;
   DATA[1439,14] := 1.0;
   DATA[1439,15] := 2.0;
   DATA[1439,16] := 1.0;
   DATA[1439,17] := 1.0;
   DATA[1439,18] := 1.0;
   DATA[1439,19] := 2.0;
   DATA[1439,20] := 148.808;
   DATA[1439,21] := 153.5247;
   DATA[1439,22] := 1.714029;
   DATA[1439,23] := 782.6839;
   DATA[1439,24] := 2.0;
   DATA[1439,25] := 2.0;
   DATA[1439,26] := 7.875737;
   DATA[1439,27] := 142.3994;
   DATA[1439,28] := 263.0095;
   DATA[1439,29] := 12.11228;
   DATA[1439,30] := 1.725968;
   DATA[1439,31] := 1.30114;
   DATA[1439,32] := 0.7352687;
   DATA[1439,33] := 0.3083624;
   DATA[1439,34] := 2.0;
   DATA[1439,35] := 250.2243;
   DATA[1439,36] := 1.649953;
   DATA[1439,37] := 189.1342;
   DATA[1439,38] := 0.000128152;
   DATA[1439,39] := 1.0;
   DATA[1440,1] := 813.1602;
   DATA[1440,2] := 1.0;
   DATA[1440,3] := 1.0;
   DATA[1440,4] := 262.5609;
   DATA[1440,5] := 8.464369;
   DATA[1440,6] := 318.3799;
   DATA[1440,8] := 1.0;
   DATA[1440,9] := 1.0;
   DATA[1440,10] := 1.0;
   DATA[1440,11] := 19.72598;
   DATA[1440,12] := 2.216571;
   DATA[1440,13] := 968.1412;
   DATA[1440,14] := 1.0;
   DATA[1440,15] := 2.0;
   DATA[1440,16] := 1.0;
   DATA[1440,17] := 1.0;
   DATA[1440,18] := 1.0;
   DATA[1440,19] := 2.0;
   DATA[1440,20] := 148.808;
   DATA[1440,21] := 153.5247;
   DATA[1440,22] := 1.714286;
   DATA[1440,23] := 783.2222;
   DATA[1440,24] := 2.0;
   DATA[1440,25] := 2.0;
   DATA[1440,26] := 7.876058;
   DATA[1440,27] := 142.3994;
   DATA[1440,28] := 263.0095;
   DATA[1440,29] := 12.11228;
   DATA[1440,30] := 1.725968;
   DATA[1440,31] := 1.292174;
   DATA[1440,32] := 0.7352687;
   DATA[1440,33] := 0.3083624;
   DATA[1440,34] := 2.0;
   DATA[1440,35] := 250.2243;
   DATA[1440,36] := 1.649953;
   DATA[1440,37] := 189.1342;
   DATA[1440,38] := 0.000128152;
   DATA[1440,39] := 1.0;
   DATA[1441,1] := 813.5527;
   DATA[1441,2] := 1.0;
   DATA[1441,3] := 1.0;
   DATA[1441,4] := 262.5609;
   DATA[1441,5] := 8.464369;
   DATA[1441,6] := 318.3799;
   DATA[1441,8] := 1.0;
   DATA[1441,9] := 1.0;
   DATA[1441,10] := 1.0;
   DATA[1441,11] := 19.72598;
   DATA[1441,12] := 2.214521;
   DATA[1441,13] := 967.9409;
   DATA[1441,14] := 1.0;
   DATA[1441,15] := 2.0;
   DATA[1441,16] := 1.0;
   DATA[1441,17] := 1.0;
   DATA[1441,18] := 1.0;
   DATA[1441,19] := 2.0;
   DATA[1441,20] := 148.808;
   DATA[1441,21] := 153.5247;
   DATA[1441,22] := 1.715311;
   DATA[1441,23] := 783.4529;
   DATA[1441,24] := 2.0;
   DATA[1441,25] := 2.0;
   DATA[1441,26] := 7.876378;
   DATA[1441,27] := 142.3994;
   DATA[1441,28] := 263.0095;
   DATA[1441,29] := 12.11228;
   DATA[1441,30] := 1.725968;
   DATA[1441,31] := 1.28372;
   DATA[1441,32] := 0.7352687;
   DATA[1441,33] := 0.3083624;
   DATA[1441,34] := 2.0;
   DATA[1441,35] := 250.2243;
   DATA[1441,36] := 1.649953;
   DATA[1441,37] := 189.1342;
   DATA[1441,38] := 0.000128152;
   DATA[1441,39] := 1.0;
   DATA[1442,1] := 813.3564;
   DATA[1442,2] := 1.0;
   DATA[1442,3] := 1.0;
   DATA[1442,4] := 262.5609;
   DATA[1442,5] := 8.464369;
   DATA[1442,6] := 318.3799;
   DATA[1442,8] := 1.0;
   DATA[1442,9] := 1.0;
   DATA[1442,10] := 1.0;
   DATA[1442,11] := 19.77399;
   DATA[1442,12] := 2.214521;
   DATA[1442,13] := 967.4603;
   DATA[1442,14] := 1.0;
   DATA[1442,15] := 2.0;
   DATA[1442,16] := 1.0;
   DATA[1442,17] := 1.0;
   DATA[1442,18] := 1.0;
   DATA[1442,19] := 2.0;
   DATA[1442,20] := 148.808;
   DATA[1442,21] := 153.5247;
   DATA[1442,22] := 1.715439;
   DATA[1442,23] := 783.6452;
   DATA[1442,24] := 2.0;
   DATA[1442,25] := 2.0;
   DATA[1442,26] := 7.876378;
   DATA[1442,27] := 142.3994;
   DATA[1442,28] := 263.0095;
   DATA[1442,29] := 12.11228;
   DATA[1442,30] := 1.725968;
   DATA[1442,31] := 1.272576;
   DATA[1442,32] := 0.7352687;
   DATA[1442,33] := 0.306761;
   DATA[1442,34] := 2.0;
   DATA[1442,35] := 250.2243;
   DATA[1442,36] := 1.649953;
   DATA[1442,37] := 189.0541;
   DATA[1442,38] := 0.000128152;
   DATA[1442,39] := 1.0;
   DATA[1443,1] := 813.5919;
   DATA[1443,2] := 1.0;
   DATA[1443,3] := 1.0;
   DATA[1443,4] := 262.5609;
   DATA[1443,5] := 8.464369;
   DATA[1443,6] := 318.3799;
   DATA[1443,8] := 1.0;
   DATA[1443,9] := 1.0;
   DATA[1443,10] := 1.0;
   DATA[1443,11] := 19.7836;
   DATA[1443,12] := 2.214521;
   DATA[1443,13] := 967.0598;
   DATA[1443,14] := 1.0;
   DATA[1443,15] := 2.0;
   DATA[1443,16] := 1.0;
   DATA[1443,17] := 1.0;
   DATA[1443,18] := 1.0;
   DATA[1443,19] := 2.0;
   DATA[1443,20] := 148.808;
   DATA[1443,21] := 153.5247;
   DATA[1443,22] := 1.715439;
   DATA[1443,23] := 783.6068;
   DATA[1443,24] := 2.0;
   DATA[1443,25] := 2.0;
   DATA[1443,26] := 7.876378;
   DATA[1443,27] := 142.3994;
   DATA[1443,28] := 263.0095;
   DATA[1443,29] := 12.11228;
   DATA[1443,30] := 1.725968;
   DATA[1443,31] := 1.271551;
   DATA[1443,32] := 0.7352687;
   DATA[1443,33] := 0.306761;
   DATA[1443,34] := 2.0;
   DATA[1443,35] := 250.2243;
   DATA[1443,36] := 1.649953;
   DATA[1443,37] := 188.8779;
   DATA[1443,38] := 0.000128152;
   DATA[1443,39] := 1.0;
   DATA[1444,1] := 813.2386;
   DATA[1444,2] := 1.0;
   DATA[1444,3] := 1.0;
   DATA[1444,4] := 262.5609;
   DATA[1444,5] := 8.464369;
   DATA[1444,6] := 318.3799;
   DATA[1444,8] := 1.0;
   DATA[1444,9] := 1.0;
   DATA[1444,10] := 1.0;
   DATA[1444,11] := 19.7836;
   DATA[1444,12] := 2.21593;
   DATA[1444,13] := 966.5391;
   DATA[1444,14] := 1.0;
   DATA[1444,15] := 2.0;
   DATA[1444,16] := 1.0;
   DATA[1444,17] := 1.0;
   DATA[1444,18] := 1.0;
   DATA[1444,19] := 2.0;
   DATA[1444,20] := 148.808;
   DATA[1444,21] := 153.5247;
   DATA[1444,22] := 1.715439;
   DATA[1444,23] := 783.6452;
   DATA[1444,24] := 2.0;
   DATA[1444,25] := 2.0;
   DATA[1444,26] := 7.876378;
   DATA[1444,27] := 142.3994;
   DATA[1444,28] := 263.0095;
   DATA[1444,29] := 12.11228;
   DATA[1444,30] := 1.723789;
   DATA[1444,31] := 1.276419;
   DATA[1444,32] := 0.7352687;
   DATA[1444,33] := 0.306761;
   DATA[1444,34] := 2.0;
   DATA[1444,35] := 250.0961;
   DATA[1444,36] := 1.649953;
   DATA[1444,37] := 188.8779;
   DATA[1444,38] := 0.000128152;
   DATA[1444,39] := 1.0;
   DATA[1445,1] := 813.0424;
   DATA[1445,2] := 1.0;
   DATA[1445,3] := 1.0;
   DATA[1445,4] := 262.5609;
   DATA[1445,5] := 8.464369;
   DATA[1445,6] := 318.3799;
   DATA[1445,8] := 1.0;
   DATA[1445,9] := 1.0;
   DATA[1445,10] := 1.0;
   DATA[1445,11] := 19.73558;
   DATA[1445,12] := 2.21593;
   DATA[1445,13] := 966.2186;
   DATA[1445,14] := 1.0;
   DATA[1445,15] := 2.0;
   DATA[1445,16] := 1.0;
   DATA[1445,17] := 1.0;
   DATA[1445,18] := 1.0;
   DATA[1445,19] := 2.0;
   DATA[1445,20] := 148.808;
   DATA[1445,21] := 153.5247;
   DATA[1445,22] := 1.713261;
   DATA[1445,23] := 783.7606;
   DATA[1445,24] := 2.0;
   DATA[1445,25] := 2.0;
   DATA[1445,26] := 7.876378;
   DATA[1445,27] := 142.3994;
   DATA[1445,28] := 263.0095;
   DATA[1445,29] := 12.11228;
   DATA[1445,30] := 1.723789;
   DATA[1445,31] := 1.291405;
   DATA[1445,32] := 0.7352687;
   DATA[1445,33] := 0.3081062;
   DATA[1445,34] := 2.0;
   DATA[1445,35] := 249.9359;
   DATA[1445,36] := 1.649953;
   DATA[1445,37] := 188.8779;
   DATA[1445,38] := 0.000128152;
   DATA[1445,39] := 1.0;
   DATA[1446,1] := 813.3171;
   DATA[1446,2] := 1.0;
   DATA[1446,3] := 1.0;
   DATA[1446,4] := 262.5609;
   DATA[1446,5] := 8.464369;
   DATA[1446,6] := 318.3799;
   DATA[1446,8] := 1.0;
   DATA[1446,9] := 1.0;
   DATA[1446,10] := 1.0;
   DATA[1446,11] := 19.73558;
   DATA[1446,12] := 2.21593;
   DATA[1446,13] := 965.4576;
   DATA[1446,14] := 1.0;
   DATA[1446,15] := 2.0;
   DATA[1446,16] := 1.0;
   DATA[1446,17] := 1.0;
   DATA[1446,18] := 1.0;
   DATA[1446,19] := 2.0;
   DATA[1446,20] := 148.808;
   DATA[1446,21] := 153.5247;
   DATA[1446,22] := 1.713261;
   DATA[1446,23] := 783.7221;
   DATA[1446,24] := 2.0;
   DATA[1446,25] := 2.0;
   DATA[1446,26] := 7.876378;
   DATA[1446,27] := 142.3994;
   DATA[1446,28] := 263.0095;
   DATA[1446,29] := 12.11228;
   DATA[1446,30] := 1.723789;
   DATA[1446,31] := 1.287562;
   DATA[1446,32] := 0.7352687;
   DATA[1446,33] := 0.3081062;
   DATA[1446,34] := 2.0;
   DATA[1446,35] := 249.9359;
   DATA[1446,36] := 1.649953;
   DATA[1446,37] := 188.8779;
   DATA[1446,38] := 0.000128152;
   DATA[1446,39] := 1.0;
   DATA[1447,1] := 813.6312;
   DATA[1447,2] := 1.0;
   DATA[1447,3] := 1.0;
   DATA[1447,4] := 262.5609;
   DATA[1447,5] := 8.464369;
   DATA[1447,6] := 318.3799;
   DATA[1447,8] := 1.0;
   DATA[1447,9] := 1.0;
   DATA[1447,10] := 1.0;
   DATA[1447,11] := 19.73558;
   DATA[1447,12] := 2.216058;
   DATA[1447,13] := 964.9769;
   DATA[1447,14] := 1.0;
   DATA[1447,15] := 2.0;
   DATA[1447,16] := 1.0;
   DATA[1447,17] := 1.0;
   DATA[1447,18] := 1.0;
   DATA[1447,19] := 2.0;
   DATA[1447,20] := 148.808;
   DATA[1447,21] := 153.6016;
   DATA[1447,22] := 1.713261;
   DATA[1447,23] := 783.799;
   DATA[1447,24] := 2.0;
   DATA[1447,25] := 2.0;
   DATA[1447,26] := 7.876378;
   DATA[1447,27] := 142.3994;
   DATA[1447,28] := 263.0095;
   DATA[1447,29] := 12.11228;
   DATA[1447,30] := 1.723789;
   DATA[1447,31] := 1.28705;
   DATA[1447,32] := 0.7352687;
   DATA[1447,33] := 0.3083624;
   DATA[1447,34] := 2.0;
   DATA[1447,35] := 249.9359;
   DATA[1447,36] := 1.649953;
   DATA[1447,37] := 188.8779;
   DATA[1447,38] := 0.000128152;
   DATA[1447,39] := 1.0;
   DATA[1448,1] := 813.5919;
   DATA[1448,2] := 1.0;
   DATA[1448,3] := 1.0;
   DATA[1448,4] := 262.5609;
   DATA[1448,5] := 8.464369;
   DATA[1448,6] := 318.3799;
   DATA[1448,8] := 1.0;
   DATA[1448,9] := 1.0;
   DATA[1448,10] := 1.0;
   DATA[1448,11] := 19.73558;
   DATA[1448,12] := 2.216827;
   DATA[1448,13] := 964.7366;
   DATA[1448,14] := 1.0;
   DATA[1448,15] := 2.0;
   DATA[1448,16] := 1.0;
   DATA[1448,17] := 1.0;
   DATA[1448,18] := 1.0;
   DATA[1448,19] := 2.0;
   DATA[1448,20] := 148.808;
   DATA[1448,21] := 153.6016;
   DATA[1448,22] := 1.713261;
   DATA[1448,23] := 783.6068;
   DATA[1448,24] := 2.0;
   DATA[1448,25] := 2.0;
   DATA[1448,26] := 7.876378;
   DATA[1448,27] := 142.3994;
   DATA[1448,28] := 263.0095;
   DATA[1448,29] := 12.11228;
   DATA[1448,30] := 1.72443;
   DATA[1448,31] := 1.291918;
   DATA[1448,32] := 0.7352687;
   DATA[1448,33] := 0.3084905;
   DATA[1448,34] := 2.0;
   DATA[1448,35] := 249.9359;
   DATA[1448,36] := 1.649953;
   DATA[1448,37] := 188.8779;
   DATA[1448,38] := 0.000128152;
   DATA[1448,39] := 1.0;
   DATA[1449,1] := 813.8275;
   DATA[1449,2] := 1.0;
   DATA[1449,3] := 1.0;
   DATA[1449,4] := 262.5609;
   DATA[1449,5] := 8.464369;
   DATA[1449,6] := 318.3799;
   DATA[1449,8] := 1.0;
   DATA[1449,9] := 1.0;
   DATA[1449,10] := 1.0;
   DATA[1449,11] := 19.73558;
   DATA[1449,12] := 2.216827;
   DATA[1449,13] := 964.3361;
   DATA[1449,14] := 1.0;
   DATA[1449,15] := 2.0;
   DATA[1449,16] := 1.0;
   DATA[1449,17] := 1.0;
   DATA[1449,18] := 1.0;
   DATA[1449,19] := 2.0;
   DATA[1449,20] := 148.808;
   DATA[1449,21] := 153.6016;
   DATA[1449,22] := 1.71467;
   DATA[1449,23] := 783.799;
   DATA[1449,24] := 2.0;
   DATA[1449,25] := 2.0;
   DATA[1449,26] := 7.876378;
   DATA[1449,27] := 142.3994;
   DATA[1449,28] := 263.0095;
   DATA[1449,29] := 12.11228;
   DATA[1449,30] := 1.724814;
   DATA[1449,31] := 1.284745;
   DATA[1449,32] := 0.7352687;
   DATA[1449,33] := 0.3084905;
   DATA[1449,34] := 2.0;
   DATA[1449,35] := 249.9359;
   DATA[1449,36] := 1.649953;
   DATA[1449,37] := 188.8779;
   DATA[1449,38] := 0.000128152;
   DATA[1449,39] := 1.0;
   DATA[1450,1] := 814.2985;
   DATA[1450,2] := 1.0;
   DATA[1450,3] := 1.0;
   DATA[1450,4] := 262.5609;
   DATA[1450,5] := 8.464369;
   DATA[1450,6] := 318.3799;
   DATA[1450,8] := 1.0;
   DATA[1450,9] := 1.0;
   DATA[1450,10] := 1.0;
   DATA[1450,11] := 19.73558;
   DATA[1450,12] := 2.218364;
   DATA[1450,13] := 963.9355;
   DATA[1450,14] := 1.0;
   DATA[1450,15] := 2.0;
   DATA[1450,16] := 1.0;
   DATA[1450,17] := 1.0;
   DATA[1450,18] := 1.0;
   DATA[1450,19] := 2.0;
   DATA[1450,20] := 148.808;
   DATA[1450,21] := 153.6016;
   DATA[1450,22] := 1.71467;
   DATA[1450,23] := 783.799;
   DATA[1450,24] := 2.0;
   DATA[1450,25] := 2.0;
   DATA[1450,26] := 7.876378;
   DATA[1450,27] := 142.3994;
   DATA[1450,28] := 263.0095;
   DATA[1450,29] := 12.11228;
   DATA[1450,30] := 1.724814;
   DATA[1450,31] := 1.28167;
   DATA[1450,32] := 0.7352687;
   DATA[1450,33] := 0.3084905;
   DATA[1450,34] := 2.0;
   DATA[1450,35] := 249.9359;
   DATA[1450,36] := 1.649953;
   DATA[1450,37] := 188.8779;
   DATA[1450,38] := 0.000128152;
   DATA[1450,39] := 1.0;
   DATA[1451,1] := 814.1022;
   DATA[1451,2] := 1.0;
   DATA[1451,3] := 1.0;
   DATA[1451,4] := 262.5609;
   DATA[1451,5] := 8.464369;
   DATA[1451,6] := 318.4055;
   DATA[1451,8] := 1.0;
   DATA[1451,9] := 1.0;
   DATA[1451,10] := 1.0;
   DATA[1451,11] := 19.73558;
   DATA[1451,12] := 2.218364;
   DATA[1451,13] := 963.4149;
   DATA[1451,14] := 1.0;
   DATA[1451,15] := 2.0;
   DATA[1451,16] := 1.0;
   DATA[1451,17] := 1.0;
   DATA[1451,18] := 1.0;
   DATA[1451,19] := 2.0;
   DATA[1451,20] := 148.808;
   DATA[1451,21] := 153.6016;
   DATA[1451,22] := 1.71467;
   DATA[1451,23] := 783.6452;
   DATA[1451,24] := 2.0;
   DATA[1451,25] := 2.0;
   DATA[1451,26] := 7.876378;
   DATA[1451,27] := 142.3994;
   DATA[1451,28] := 263.0095;
   DATA[1451,29] := 12.11228;
   DATA[1451,30] := 1.724814;
   DATA[1451,31] := 1.271935;
   DATA[1451,32] := 0.7352687;
   DATA[1451,33] := 0.3084905;
   DATA[1451,34] := 2.0;
   DATA[1451,35] := 249.9359;
   DATA[1451,36] := 1.649953;
   DATA[1451,37] := 188.7817;
   DATA[1451,38] := 0.000128152;
   DATA[1451,39] := 1.0;
   DATA[1452,1] := 814.0237;
   DATA[1452,2] := 1.0;
   DATA[1452,3] := 1.0;
   DATA[1452,4] := 262.5609;
   DATA[1452,5] := 8.464369;
   DATA[1452,6] := 318.5594;
   DATA[1452,8] := 1.0;
   DATA[1452,9] := 1.0;
   DATA[1452,10] := 1.0;
   DATA[1452,11] := 19.73558;
   DATA[1452,12] := 2.218364;
   DATA[1452,13] := 963.1745;
   DATA[1452,14] := 1.0;
   DATA[1452,15] := 2.0;
   DATA[1452,16] := 1.0;
   DATA[1452,17] := 1.0;
   DATA[1452,18] := 1.0;
   DATA[1452,19] := 2.0;
   DATA[1452,20] := 148.808;
   DATA[1452,21] := 153.6016;
   DATA[1452,22] := 1.715824;
   DATA[1452,23] := 784.1066;
   DATA[1452,24] := 2.0;
   DATA[1452,25] := 2.0;
   DATA[1452,26] := 7.876378;
   DATA[1452,27] := 142.3994;
   DATA[1452,28] := 263.0095;
   DATA[1452,29] := 12.11228;
   DATA[1452,30] := 1.724814;
   DATA[1452,31] := 1.262329;
   DATA[1452,32] := 0.7352687;
   DATA[1452,33] := 0.3084905;
   DATA[1452,34] := 2.0;
   DATA[1452,35] := 249.9359;
   DATA[1452,36] := 1.649953;
   DATA[1452,37] := 188.7817;
   DATA[1452,38] := 0.000128152;
   DATA[1452,39] := 1.0;
   DATA[1453,1] := 813.9844;
   DATA[1453,2] := 1.0;
   DATA[1453,3] := 1.0;
   DATA[1453,4] := 262.5609;
   DATA[1453,5] := 8.464369;
   DATA[1453,6] := 318.5594;
   DATA[1453,8] := 1.0;
   DATA[1453,9] := 1.0;
   DATA[1453,10] := 1.0;
   DATA[1453,11] := 19.75799;
   DATA[1453,12] := 2.218364;
   DATA[1453,13] := 962.7339;
   DATA[1453,14] := 1.0;
   DATA[1453,15] := 2.0;
   DATA[1453,16] := 1.0;
   DATA[1453,17] := 1.0;
   DATA[1453,18] := 1.0;
   DATA[1453,19] := 2.0;
   DATA[1453,20] := 148.808;
   DATA[1453,21] := 153.6016;
   DATA[1453,22] := 1.71608;
   DATA[1453,23] := 783.9913;
   DATA[1453,24] := 2.0;
   DATA[1453,25] := 2.0;
   DATA[1453,26] := 7.876378;
   DATA[1453,27] := 142.3994;
   DATA[1453,28] := 263.0095;
   DATA[1453,29] := 12.11228;
   DATA[1453,30] := 1.723789;
   DATA[1453,31] := 1.269374;
   DATA[1453,32] := 0.7352687;
   DATA[1453,33] := 0.3084905;
   DATA[1453,34] := 2.0;
   DATA[1453,35] := 249.9359;
   DATA[1453,36] := 1.649953;
   DATA[1453,37] := 188.7817;
   DATA[1453,38] := 0.000128152;
   DATA[1453,39] := 1.0;
   DATA[1454,1] := 814.22;
   DATA[1454,2] := 1.0;
   DATA[1454,3] := 1.0;
   DATA[1454,4] := 262.5609;
   DATA[1454,5] := 8.464369;
   DATA[1454,6] := 318.5594;
   DATA[1454,8] := 1.0;
   DATA[1454,9] := 1.0;
   DATA[1454,10] := 1.0;
   DATA[1454,11] := 19.7836;
   DATA[1454,12] := 2.218364;
   DATA[1454,13] := 961.7326;
   DATA[1454,14] := 1.0;
   DATA[1454,15] := 2.0;
   DATA[1454,16] := 1.0;
   DATA[1454,17] := 1.0;
   DATA[1454,18] := 1.0;
   DATA[1454,19] := 2.0;
   DATA[1454,20] := 148.808;
   DATA[1454,21] := 153.6016;
   DATA[1454,22] := 1.71608;
   DATA[1454,23] := 783.9528;
   DATA[1454,24] := 2.0;
   DATA[1454,25] := 2.0;
   DATA[1454,26] := 7.876378;
   DATA[1454,27] := 142.3994;
   DATA[1454,28] := 263.0095;
   DATA[1454,29] := 12.11228;
   DATA[1454,30] := 1.723789;
   DATA[1454,31] := 1.271935;
   DATA[1454,32] := 0.7352687;
   DATA[1454,33] := 0.3084905;
   DATA[1454,34] := 2.0;
   DATA[1454,35] := 249.9359;
   DATA[1454,36] := 1.649953;
   DATA[1454,37] := 188.7817;
   DATA[1454,38] := 0.000128152;
   DATA[1454,39] := 1.0;
   DATA[1455,1] := 813.9844;
   DATA[1455,2] := 1.0;
   DATA[1455,3] := 1.0;
   DATA[1455,4] := 262.5609;
   DATA[1455,5] := 8.464369;
   DATA[1455,6] := 318.5594;
   DATA[1455,8] := 1.0;
   DATA[1455,9] := 1.0;
   DATA[1455,10] := 1.0;
   DATA[1455,11] := 19.7836;
   DATA[1455,12] := 2.218364;
   DATA[1455,13] := 961.1718;
   DATA[1455,14] := 1.0;
   DATA[1455,15] := 2.0;
   DATA[1455,16] := 1.0;
   DATA[1455,17] := 1.0;
   DATA[1455,18] := 1.0;
   DATA[1455,19] := 2.0;
   DATA[1455,20] := 148.808;
   DATA[1455,21] := 153.6016;
   DATA[1455,22] := 1.71608;
   DATA[1455,23] := 783.6452;
   DATA[1455,24] := 2.0;
   DATA[1455,25] := 2.0;
   DATA[1455,26] := 7.876378;
   DATA[1455,27] := 142.3994;
   DATA[1455,28] := 263.0095;
   DATA[1455,29] := 12.11228;
   DATA[1455,30] := 1.723789;
   DATA[1455,31] := 1.271935;
   DATA[1455,32] := 0.7352687;
   DATA[1455,33] := 0.3084905;
   DATA[1455,34] := 2.0;
   DATA[1455,35] := 249.9359;
   DATA[1455,36] := 1.649953;
   DATA[1455,37] := 188.7817;
   DATA[1455,38] := 0.000128152;
   DATA[1455,39] := 1.0;
   DATA[1456,1] := 813.8275;
   DATA[1456,2] := 1.0;
   DATA[1456,3] := 1.0;
   DATA[1456,4] := 262.5609;
   DATA[1456,5] := 8.464369;
   DATA[1456,6] := 318.5594;
   DATA[1456,8] := 1.0;
   DATA[1456,9] := 1.0;
   DATA[1456,10] := 1.0;
   DATA[1456,11] := 19.68436;
   DATA[1456,12] := 2.218364;
   DATA[1456,13] := 960.7713;
   DATA[1456,14] := 1.0;
   DATA[1456,15] := 2.0;
   DATA[1456,16] := 1.0;
   DATA[1456,17] := 1.0;
   DATA[1456,18] := 1.0;
   DATA[1456,19] := 2.0;
   DATA[1456,20] := 148.808;
   DATA[1456,21] := 153.6016;
   DATA[1456,22] := 1.714158;
   DATA[1456,23] := 783.7606;
   DATA[1456,24] := 2.0;
   DATA[1456,25] := 2.0;
   DATA[1456,26] := 7.876378;
   DATA[1456,27] := 142.3994;
   DATA[1456,28] := 263.0095;
   DATA[1456,29] := 12.11228;
   DATA[1456,30] := 1.723789;
   DATA[1456,31] := 1.287434;
   DATA[1456,32] := 0.7352687;
   DATA[1456,33] := 0.3084905;
   DATA[1456,34] := 2.0;
   DATA[1456,35] := 249.984;
   DATA[1456,36] := 1.649953;
   DATA[1456,37] := 188.7817;
   DATA[1456,38] := 0.000128152;
   DATA[1456,39] := 1.0;
   DATA[1457,1] := 813.7489;
   DATA[1457,2] := 1.0;
   DATA[1457,3] := 1.0;
   DATA[1457,4] := 262.5609;
   DATA[1457,5] := 8.464369;
   DATA[1457,6] := 318.5594;
   DATA[1457,8] := 1.0;
   DATA[1457,9] := 1.0;
   DATA[1457,10] := 1.0;
   DATA[1457,11] := 19.64274;
   DATA[1457,12] := 2.218364;
   DATA[1457,13] := 960.1705;
   DATA[1457,14] := 1.0;
   DATA[1457,15] := 2.0;
   DATA[1457,16] := 1.0;
   DATA[1457,17] := 1.0;
   DATA[1457,18] := 1.0;
   DATA[1457,19] := 2.0;
   DATA[1457,20] := 148.808;
   DATA[1457,21] := 153.6016;
   DATA[1457,22] := 1.713261;
   DATA[1457,23] := 784.2989;
   DATA[1457,24] := 2.0;
   DATA[1457,25] := 2.0;
   DATA[1457,26] := 7.876378;
   DATA[1457,27] := 142.3994;
   DATA[1457,28] := 263.0095;
   DATA[1457,29] := 12.11228;
   DATA[1457,30] := 1.723789;
   DATA[1457,31] := 1.285001;
   DATA[1457,32] := 0.7352687;
   DATA[1457,33] := 0.3106684;
   DATA[1457,34] := 2.0;
   DATA[1457,35] := 250.0641;
   DATA[1457,36] := 1.649953;
   DATA[1457,37] := 188.7817;
   DATA[1457,38] := 0.000128152;
   DATA[1457,39] := 1.0;
   DATA[1458,1] := 813.7097;
   DATA[1458,2] := 1.0;
   DATA[1458,3] := 1.0;
   DATA[1458,4] := 262.5609;
   DATA[1458,5] := 8.464369;
   DATA[1458,6] := 318.5594;
   DATA[1458,8] := 1.0;
   DATA[1458,9] := 1.0;
   DATA[1458,10] := 1.0;
   DATA[1458,11] := 19.64274;
   DATA[1458,12] := 2.218364;
   DATA[1458,13] := 960.1304;
   DATA[1458,14] := 1.0;
   DATA[1458,15] := 2.0;
   DATA[1458,16] := 1.0;
   DATA[1458,17] := 1.0;
   DATA[1458,18] := 1.0;
   DATA[1458,19] := 2.0;
   DATA[1458,20] := 148.808;
   DATA[1458,21] := 153.6016;
   DATA[1458,22] := 1.713261;
   DATA[1458,23] := 784.1066;
   DATA[1458,24] := 2.0;
   DATA[1458,25] := 2.0;
   DATA[1458,26] := 7.876378;
   DATA[1458,27] := 142.3994;
   DATA[1458,28] := 263.0095;
   DATA[1458,29] := 12.11228;
   DATA[1458,30] := 1.723789;
   DATA[1458,31] := 1.285001;
   DATA[1458,32] := 0.7352687;
   DATA[1458,33] := 0.3106684;
   DATA[1458,34] := 2.0;
   DATA[1458,35] := 250.0641;
   DATA[1458,36] := 1.649953;
   DATA[1458,37] := 188.7817;
   DATA[1458,38] := 0.000128152;
   DATA[1458,39] := 1.0;
   DATA[1459,1] := 813.9059;
   DATA[1459,2] := 1.0;
   DATA[1459,3] := 1.0;
   DATA[1459,4] := 262.5609;
   DATA[1459,5] := 8.464369;
   DATA[1459,6] := 318.5594;
   DATA[1459,8] := 1.0;
   DATA[1459,9] := 1.0;
   DATA[1459,10] := 1.0;
   DATA[1459,11] := 19.64274;
   DATA[1459,12] := 2.214009;
   DATA[1459,13] := 959.2893;
   DATA[1459,14] := 1.0;
   DATA[1459,15] := 2.0;
   DATA[1459,16] := 1.0;
   DATA[1459,17] := 1.0;
   DATA[1459,18] := 1.0;
   DATA[1459,19] := 2.0;
   DATA[1459,20] := 148.808;
   DATA[1459,21] := 153.6016;
   DATA[1459,22] := 1.713261;
   DATA[1459,23] := 784.2989;
   DATA[1459,24] := 2.0;
   DATA[1459,25] := 2.0;
   DATA[1459,26] := 7.876378;
   DATA[1459,27] := 142.3994;
   DATA[1459,28] := 263.0095;
   DATA[1459,29] := 12.11228;
   DATA[1459,30] := 1.723789;
   DATA[1459,31] := 1.300372;
   DATA[1459,32] := 0.7352687;
   DATA[1459,33] := 0.3106684;
   DATA[1459,34] := 2.0;
   DATA[1459,35] := 250.0641;
   DATA[1459,36] := 1.649953;
   DATA[1459,37] := 188.8458;
   DATA[1459,38] := 0.000128152;
   DATA[1459,39] := 1.0;
   DATA[1460,1] := 813.8275;
   DATA[1460,2] := 1.0;
   DATA[1460,3] := 1.0;
   DATA[1460,4] := 262.5609;
   DATA[1460,5] := 8.464369;
   DATA[1460,6] := 318.5594;
   DATA[1460,8] := 1.0;
   DATA[1460,9] := 1.0;
   DATA[1460,10] := 1.0;
   DATA[1460,11] := 19.70677;
   DATA[1460,12] := 2.214009;
   DATA[1460,13] := 958.5283;
   DATA[1460,14] := 1.0;
   DATA[1460,15] := 2.0;
   DATA[1460,16] := 1.0;
   DATA[1460,17] := 1.0;
   DATA[1460,18] := 1.0;
   DATA[1460,19] := 2.0;
   DATA[1460,20] := 148.808;
   DATA[1460,21] := 153.6016;
   DATA[1460,22] := 1.713261;
   DATA[1460,23] := 784.5296;
   DATA[1460,24] := 2.0;
   DATA[1460,25] := 2.0;
   DATA[1460,26] := 7.876378;
   DATA[1460,27] := 142.3994;
   DATA[1460,28] := 263.0095;
   DATA[1460,29] := 12.11228;
   DATA[1460,30] := 1.723789;
   DATA[1460,31] := 1.291918;
   DATA[1460,32] := 0.7352687;
   DATA[1460,33] := 0.3106684;
   DATA[1460,34] := 2.0;
   DATA[1460,35] := 250.0641;
   DATA[1460,36] := 1.649953;
   DATA[1460,37] := 188.8458;
   DATA[1460,38] := 0.000128152;
   DATA[1460,39] := 1.0;
   DATA[1461,1] := 813.7489;
   DATA[1461,2] := 1.0;
   DATA[1461,3] := 1.0;
   DATA[1461,4] := 262.5609;
   DATA[1461,5] := 8.464369;
   DATA[1461,6] := 318.5594;
   DATA[1461,8] := 1.0;
   DATA[1461,9] := 1.0;
   DATA[1461,10] := 1.0;
   DATA[1461,11] := 19.70677;
   DATA[1461,12] := 2.214009;
   DATA[1461,13] := 957.6071;
   DATA[1461,14] := 1.0;
   DATA[1461,15] := 2.0;
   DATA[1461,16] := 1.0;
   DATA[1461,17] := 1.0;
   DATA[1461,18] := 1.0;
   DATA[1461,19] := 2.0;
   DATA[1461,20] := 148.808;
   DATA[1461,21] := 153.6016;
   DATA[1461,22] := 1.713261;
   DATA[1461,23] := 784.6834;
   DATA[1461,24] := 2.0;
   DATA[1461,25] := 2.0;
   DATA[1461,26] := 7.876378;
   DATA[1461,27] := 142.3994;
   DATA[1461,28] := 263.0095;
   DATA[1461,29] := 12.11228;
   DATA[1461,30] := 1.723789;
   DATA[1461,31] := 1.290893;
   DATA[1461,32] := 0.7352687;
   DATA[1461,33] := 0.3106684;
   DATA[1461,34] := 2.0;
   DATA[1461,35] := 250.0641;
   DATA[1461,36] := 1.649953;
   DATA[1461,37] := 188.8458;
   DATA[1461,38] := 0.000128152;
   DATA[1461,39] := 1.0;
   DATA[1462,1] := 813.9844;
   DATA[1462,2] := 1.0;
   DATA[1462,3] := 1.0;
   DATA[1462,4] := 262.5609;
   DATA[1462,5] := 8.464369;
   DATA[1462,6] := 318.5594;
   DATA[1462,8] := 1.0;
   DATA[1462,9] := 1.0;
   DATA[1462,10] := 1.0;
   DATA[1462,11] := 19.70677;
   DATA[1462,12] := 2.214009;
   DATA[1462,13] := 957.3667;
   DATA[1462,14] := 1.0;
   DATA[1462,15] := 2.0;
   DATA[1462,16] := 1.0;
   DATA[1462,17] := 1.0;
   DATA[1462,18] := 1.0;
   DATA[1462,19] := 2.0;
   DATA[1462,20] := 148.808;
   DATA[1462,21] := 153.6016;
   DATA[1462,22] := 1.713261;
   DATA[1462,23] := 784.7988;
   DATA[1462,24] := 2.0;
   DATA[1462,25] := 2.0;
   DATA[1462,26] := 7.876378;
   DATA[1462,27] := 142.3994;
   DATA[1462,28] := 263.0095;
   DATA[1462,29] := 12.11228;
   DATA[1462,30] := 1.722763;
   DATA[1462,31] := 1.28167;
   DATA[1462,32] := 0.7352687;
   DATA[1462,33] := 0.3106684;
   DATA[1462,34] := 2.0;
   DATA[1462,35] := 250.0641;
   DATA[1462,36] := 1.649953;
   DATA[1462,37] := 188.8458;
   DATA[1462,38] := 0.000128152;
   DATA[1462,39] := 1.0;
   DATA[1463,1] := 814.1415;
   DATA[1463,2] := 1.0;
   DATA[1463,3] := 1.0;
   DATA[1463,4] := 262.5609;
   DATA[1463,5] := 8.464369;
   DATA[1463,6] := 318.5594;
   DATA[1463,8] := 1.0;
   DATA[1463,9] := 1.0;
   DATA[1463,10] := 1.0;
   DATA[1463,11] := 19.70677;
   DATA[1463,12] := 2.214009;
   DATA[1463,13] := 956.9261;
   DATA[1463,14] := 1.0;
   DATA[1463,15] := 2.0;
   DATA[1463,16] := 1.0;
   DATA[1463,17] := 1.0;
   DATA[1463,18] := 1.0;
   DATA[1463,19] := 2.0;
   DATA[1463,20] := 148.808;
   DATA[1463,21] := 153.6016;
   DATA[1463,22] := 1.713261;
   DATA[1463,23] := 784.6834;
   DATA[1463,24] := 2.0;
   DATA[1463,25] := 2.0;
   DATA[1463,26] := 7.876378;
   DATA[1463,27] := 142.3994;
   DATA[1463,28] := 263.0095;
   DATA[1463,29] := 12.11228;
   DATA[1463,30] := 1.722763;
   DATA[1463,31] := 1.280902;
   DATA[1463,32] := 0.7352687;
   DATA[1463,33] := 0.3093873;
   DATA[1463,34] := 2.0;
   DATA[1463,35] := 250.0641;
   DATA[1463,36] := 1.649953;
   DATA[1463,37] := 188.8939;
   DATA[1463,38] := 0.000128152;
   DATA[1463,39] := 1.0;
   DATA[1464,1] := 814.1022;
   DATA[1464,2] := 1.0;
   DATA[1464,3] := 1.0;
   DATA[1464,4] := 262.5609;
   DATA[1464,5] := 8.464369;
   DATA[1464,6] := 318.5594;
   DATA[1464,8] := 1.0;
   DATA[1464,9] := 1.0;
   DATA[1464,10] := 1.0;
   DATA[1464,11] := 19.75479;
   DATA[1464,12] := 2.214009;
   DATA[1464,13] := 956.5256;
   DATA[1464,14] := 1.0;
   DATA[1464,15] := 2.0;
   DATA[1464,16] := 1.0;
   DATA[1464,17] := 1.0;
   DATA[1464,18] := 1.0;
   DATA[1464,19] := 2.0;
   DATA[1464,20] := 148.808;
   DATA[1464,21] := 153.6016;
   DATA[1464,22] := 1.713261;
   DATA[1464,23] := 784.9141;
   DATA[1464,24] := 2.0;
   DATA[1464,25] := 2.0;
   DATA[1464,26] := 7.876378;
   DATA[1464,27] := 142.3994;
   DATA[1464,28] := 263.0095;
   DATA[1464,29] := 12.11228;
   DATA[1464,30] := 1.721866;
   DATA[1464,31] := 1.290252;
   DATA[1464,32] := 0.7352687;
   DATA[1464,33] := 0.3088108;
   DATA[1464,34] := 2.0;
   DATA[1464,35] := 250.0641;
   DATA[1464,36] := 1.649953;
   DATA[1464,37] := 189.006;
   DATA[1464,38] := 0.000128152;
   DATA[1464,39] := 1.0;
   DATA[1465,1] := 813.7882;
   DATA[1465,2] := 1.0;
   DATA[1465,3] := 1.0;
   DATA[1465,4] := 262.5609;
   DATA[1465,5] := 8.464369;
   DATA[1465,6] := 318.5594;
   DATA[1465,8] := 1.0;
   DATA[1465,9] := 1.0;
   DATA[1465,10] := 1.0;
   DATA[1465,11] := 19.7964;
   DATA[1465,12] := 2.214009;
   DATA[1465,13] := 955.9648;
   DATA[1465,14] := 1.0;
   DATA[1465,15] := 2.0;
   DATA[1465,16] := 1.0;
   DATA[1465,17] := 1.0;
   DATA[1465,18] := 1.0;
   DATA[1465,19] := 2.0;
   DATA[1465,20] := 148.808;
   DATA[1465,21] := 153.6016;
   DATA[1465,22] := 1.713261;
   DATA[1465,23] := 784.8757;
   DATA[1465,24] := 2.0;
   DATA[1465,25] := 2.0;
   DATA[1465,26] := 7.876378;
   DATA[1465,27] := 142.3994;
   DATA[1465,28] := 263.0095;
   DATA[1465,29] := 12.11228;
   DATA[1465,30] := 1.72161;
   DATA[1465,31] := 1.295376;
   DATA[1465,32] := 0.7352687;
   DATA[1465,33] := 0.3084905;
   DATA[1465,34] := 2.0;
   DATA[1465,35] := 250.0641;
   DATA[1465,36] := 1.649953;
   DATA[1465,37] := 189.006;
   DATA[1465,38] := 0.000128152;
   DATA[1465,39] := 1.0;
   DATA[1466,1] := 813.7882;
   DATA[1466,2] := 1.0;
   DATA[1466,3] := 1.0;
   DATA[1466,4] := 262.5609;
   DATA[1466,5] := 8.464369;
   DATA[1466,6] := 318.5594;
   DATA[1466,8] := 1.0;
   DATA[1466,9] := 1.0;
   DATA[1466,10] := 1.0;
   DATA[1466,11] := 19.7964;
   DATA[1466,12] := 2.214009;
   DATA[1466,13] := 955.6044;
   DATA[1466,14] := 1.0;
   DATA[1466,15] := 2.0;
   DATA[1466,16] := 1.0;
   DATA[1466,17] := 1.0;
   DATA[1466,18] := 1.0;
   DATA[1466,19] := 2.0;
   DATA[1466,20] := 148.808;
   DATA[1466,21] := 153.6016;
   DATA[1466,22] := 1.713261;
   DATA[1466,23] := 785.3755;
   DATA[1466,24] := 2.0;
   DATA[1466,25] := 2.0;
   DATA[1466,26] := 7.876378;
   DATA[1466,27] := 142.3994;
   DATA[1466,28] := 263.1377;
   DATA[1466,29] := 12.11228;
   DATA[1466,30] := 1.72161;
   DATA[1466,31] := 1.301396;
   DATA[1466,32] := 0.7352687;
   DATA[1466,33] := 0.3084905;
   DATA[1466,34] := 2.0;
   DATA[1466,35] := 250.0641;
   DATA[1466,36] := 1.649953;
   DATA[1466,37] := 188.7176;
   DATA[1466,38] := 0.000128152;
   DATA[1466,39] := 1.0;
   DATA[1467,1] := 814.0237;
   DATA[1467,2] := 1.0;
   DATA[1467,3] := 1.0;
   DATA[1467,4] := 262.5609;
   DATA[1467,5] := 8.464369;
   DATA[1467,6] := 318.5594;
   DATA[1467,8] := 1.0;
   DATA[1467,9] := 1.0;
   DATA[1467,10] := 1.0;
   DATA[1467,11] := 19.77079;
   DATA[1467,12] := 2.214009;
   DATA[1467,13] := 955.1638;
   DATA[1467,14] := 1.0;
   DATA[1467,15] := 2.0;
   DATA[1467,16] := 1.0;
   DATA[1467,17] := 1.0;
   DATA[1467,18] := 1.0;
   DATA[1467,19] := 2.0;
   DATA[1467,20] := 148.808;
   DATA[1467,21] := 153.6016;
   DATA[1467,22] := 1.713261;
   DATA[1467,23] := 785.2986;
   DATA[1467,24] := 2.0;
   DATA[1467,25] := 2.0;
   DATA[1467,26] := 7.876378;
   DATA[1467,27] := 142.3994;
   DATA[1467,28] := 263.2018;
   DATA[1467,29] := 12.11228;
   DATA[1467,30] := 1.72161;
   DATA[1467,31] := 1.293711;
   DATA[1467,32] := 0.7352687;
   DATA[1467,33] := 0.3084905;
   DATA[1467,34] := 2.0;
   DATA[1467,35] := 249.8718;
   DATA[1467,36] := 1.649953;
   DATA[1467,37] := 188.7176;
   DATA[1467,38] := 0.000128152;
   DATA[1467,39] := 1.0;
   DATA[1468,1] := 813.7097;
   DATA[1468,2] := 1.0;
   DATA[1468,3] := 1.0;
   DATA[1468,4] := 262.5609;
   DATA[1468,5] := 8.464369;
   DATA[1468,6] := 318.5594;
   DATA[1468,8] := 1.0;
   DATA[1468,9] := 1.0;
   DATA[1468,10] := 1.0;
   DATA[1468,11] := 19.74838;
   DATA[1468,12] := 2.216187;
   DATA[1468,13] := 955.2038;
   DATA[1468,14] := 1.0;
   DATA[1468,15] := 2.0;
   DATA[1468,16] := 1.0;
   DATA[1468,17] := 1.0;
   DATA[1468,18] := 1.0;
   DATA[1468,19] := 2.0;
   DATA[1468,20] := 148.808;
   DATA[1468,21] := 153.294;
   DATA[1468,22] := 1.711723;
   DATA[1468,23] := 785.1833;
   DATA[1468,24] := 2.0;
   DATA[1468,25] := 2.0;
   DATA[1468,26] := 7.876378;
   DATA[1468,27] := 142.3994;
   DATA[1468,28] := 263.2018;
   DATA[1468,29] := 12.11228;
   DATA[1468,30] := 1.72161;
   DATA[1468,31] := 1.290765;
   DATA[1468,32] := 0.7352687;
   DATA[1468,33] := 0.3083624;
   DATA[1468,34] := 2.0;
   DATA[1468,35] := 249.7597;
   DATA[1468,36] := 1.649953;
   DATA[1468,37] := 188.7176;
   DATA[1468,38] := 0.000128152;
   DATA[1468,39] := 1.0;
   DATA[1469,1] := 813.6312;
   DATA[1469,2] := 1.0;
   DATA[1469,3] := 1.0;
   DATA[1469,4] := 262.5609;
   DATA[1469,5] := 8.464369;
   DATA[1469,6] := 318.5594;
   DATA[1469,8] := 1.0;
   DATA[1469,9] := 1.0;
   DATA[1469,10] := 1.0;
   DATA[1469,11] := 19.70997;
   DATA[1469,12] := 2.21798;
   DATA[1469,13] := 955.2839;
   DATA[1469,14] := 1.0;
   DATA[1469,15] := 2.0;
   DATA[1469,16] := 1.0;
   DATA[1469,17] := 1.0;
   DATA[1469,18] := 1.0;
   DATA[1469,19] := 2.0;
   DATA[1469,20] := 148.808;
   DATA[1469,21] := 153.294;
   DATA[1469,22] := 1.711723;
   DATA[1469,23] := 784.991;
   DATA[1469,24] := 2.0;
   DATA[1469,25] := 2.0;
   DATA[1469,26] := 7.876378;
   DATA[1469,27] := 142.3994;
   DATA[1469,28] := 263.2018;
   DATA[1469,29] := 12.11228;
   DATA[1469,30] := 1.72161;
   DATA[1469,31] := 1.290765;
   DATA[1469,32] := 0.7352687;
   DATA[1469,33] := 0.3083624;
   DATA[1469,34] := 2.0;
   DATA[1469,35] := 249.7597;
   DATA[1469,36] := 1.649953;
   DATA[1469,37] := 188.6055;
   DATA[1469,38] := 0.000128152;
   DATA[1469,39] := 1.0;
   DATA[1470,1] := 813.5919;
   DATA[1470,2] := 1.0;
   DATA[1470,3] := 1.0;
   DATA[1470,4] := 262.5609;
   DATA[1470,5] := 8.464369;
   DATA[1470,6] := 318.5594;
   DATA[1470,8] := 1.0;
   DATA[1470,9] := 1.0;
   DATA[1470,10] := 1.0;
   DATA[1470,11] := 19.70357;
   DATA[1470,12] := 2.219133;
   DATA[1470,13] := 954.9235;
   DATA[1470,14] := 1.0;
   DATA[1470,15] := 2.0;
   DATA[1470,16] := 1.0;
   DATA[1470,17] := 1.0;
   DATA[1470,18] := 1.0;
   DATA[1470,19] := 2.0;
   DATA[1470,20] := 148.808;
   DATA[1470,21] := 153.294;
   DATA[1470,22] := 1.711723;
   DATA[1470,23] := 785.3371;
   DATA[1470,24] := 2.0;
   DATA[1470,25] := 2.0;
   DATA[1470,26] := 7.876378;
   DATA[1470,27] := 142.3994;
   DATA[1470,28] := 263.2018;
   DATA[1470,29] := 12.11228;
   DATA[1470,30] := 1.720456;
   DATA[1470,31] := 1.290765;
   DATA[1470,32] := 0.7352687;
   DATA[1470,33] := 0.3083624;
   DATA[1470,34] := 2.0;
   DATA[1470,35] := 249.6635;
   DATA[1470,36] := 1.649953;
   DATA[1470,37] := 188.5414;
   DATA[1470,38] := 0.000128152;
   DATA[1470,39] := 1.0;
   DATA[1471,1] := 813.5919;
   DATA[1471,2] := 1.0;
   DATA[1471,3] := 1.0;
   DATA[1471,4] := 262.5609;
   DATA[1471,5] := 8.464369;
   DATA[1471,6] := 318.5594;
   DATA[1471,8] := 1.0;
   DATA[1471,9] := 1.0;
   DATA[1471,10] := 1.0;
   DATA[1471,11] := 19.70357;
   DATA[1471,12] := 2.219133;
   DATA[1471,13] := 954.9235;
   DATA[1471,14] := 1.0;
   DATA[1471,15] := 2.0;
   DATA[1471,16] := 1.0;
   DATA[1471,17] := 1.0;
   DATA[1471,18] := 1.0;
   DATA[1471,19] := 2.0;
   DATA[1471,20] := 148.808;
   DATA[1471,21] := 153.294;
   DATA[1471,22] := 1.711723;
   DATA[1471,23] := 785.3371;
   DATA[1471,24] := 2.0;
   DATA[1471,25] := 2.0;
   DATA[1471,26] := 7.876378;
   DATA[1471,27] := 142.3994;
   DATA[1471,28] := 263.2018;
   DATA[1471,29] := 12.11228;
   DATA[1471,30] := 1.720456;
   DATA[1471,31] := 1.290765;
   DATA[1471,32] := 0.7352687;
   DATA[1471,33] := 0.3083624;
   DATA[1471,34] := 2.0;
   DATA[1471,35] := 249.6635;
   DATA[1471,36] := 1.649953;
   DATA[1471,37] := 188.5414;
   DATA[1471,38] := 0.000128152;
   DATA[1471,39] := 1.0;
   DATA[1472,1] := 813.5919;
   DATA[1472,2] := 1.0;
   DATA[1472,3] := 1.0;
   DATA[1472,4] := 262.5609;
   DATA[1472,5] := 8.464369;
   DATA[1472,6] := 318.5594;
   DATA[1472,8] := 1.0;
   DATA[1472,9] := 1.0;
   DATA[1472,10] := 1.0;
   DATA[1472,11] := 19.70357;
   DATA[1472,12] := 2.219133;
   DATA[1472,13] := 954.5629;
   DATA[1472,14] := 1.0;
   DATA[1472,15] := 2.0;
   DATA[1472,16] := 1.0;
   DATA[1472,17] := 1.0;
   DATA[1472,18] := 1.0;
   DATA[1472,19] := 2.0;
   DATA[1472,20] := 148.808;
   DATA[1472,21] := 153.294;
   DATA[1472,22] := 1.711723;
   DATA[1472,23] := 785.5294;
   DATA[1472,24] := 2.0;
   DATA[1472,25] := 2.0;
   DATA[1472,26] := 7.876378;
   DATA[1472,27] := 142.3994;
   DATA[1472,28] := 263.0095;
   DATA[1472,29] := 12.11228;
   DATA[1472,30] := 1.720456;
   DATA[1472,31] := 1.290893;
   DATA[1472,32] := 0.7352687;
   DATA[1472,33] := 0.3083624;
   DATA[1472,34] := 2.0;
   DATA[1472,35] := 249.6635;
   DATA[1472,36] := 1.649953;
   DATA[1472,37] := 188.5414;
   DATA[1472,38] := 0.000128152;
   DATA[1472,39] := 1.0;
   DATA[1473,1] := 813.5134;
   DATA[1473,2] := 1.0;
   DATA[1473,3] := 1.0;
   DATA[1473,4] := 262.5609;
   DATA[1473,5] := 8.464369;
   DATA[1473,6] := 318.5594;
   DATA[1473,8] := 1.0;
   DATA[1473,9] := 1.0;
   DATA[1473,10] := 1.0;
   DATA[1473,11] := 19.72598;
   DATA[1473,12] := 2.218108;
   DATA[1473,13] := 953.4014;
   DATA[1473,14] := 1.0;
   DATA[1473,15] := 2.0;
   DATA[1473,16] := 1.0;
   DATA[1473,17] := 1.0;
   DATA[1473,18] := 1.0;
   DATA[1473,19] := 2.0;
   DATA[1473,20] := 148.808;
   DATA[1473,21] := 153.3709;
   DATA[1473,22] := 1.711723;
   DATA[1473,23] := 785.5678;
   DATA[1473,24] := 2.0;
   DATA[1473,25] := 2.0;
   DATA[1473,26] := 7.876378;
   DATA[1473,27] := 142.3994;
   DATA[1473,28] := 263.0095;
   DATA[1473,29] := 12.11228;
   DATA[1473,30] := 1.720456;
   DATA[1473,31] := 1.291789;
   DATA[1473,32] := 0.7352687;
   DATA[1473,33] := 0.3106043;
   DATA[1473,34] := 2.0;
   DATA[1473,35] := 249.7917;
   DATA[1473,36] := 1.730048;
   DATA[1473,37] := 188.5414;
   DATA[1473,38] := 0.000128152;
   DATA[1473,39] := 1.0;
   DATA[1474,1] := 813.7097;
   DATA[1474,2] := 1.0;
   DATA[1474,3] := 1.0;
   DATA[1474,4] := 262.5609;
   DATA[1474,5] := 8.464369;
   DATA[1474,6] := 318.4312;
   DATA[1474,8] := 1.0;
   DATA[1474,9] := 1.0;
   DATA[1474,10] := 1.0;
   DATA[1474,11] := 19.74838;
   DATA[1474,12] := 2.218108;
   DATA[1474,13] := 953.2813;
   DATA[1474,14] := 1.0;
   DATA[1474,15] := 2.0;
   DATA[1474,16] := 1.0;
   DATA[1474,17] := 1.0;
   DATA[1474,18] := 1.0;
   DATA[1474,19] := 2.0;
   DATA[1474,20] := 148.808;
   DATA[1474,21] := 153.3709;
   DATA[1474,22] := 1.711723;
   DATA[1474,23] := 785.5678;
   DATA[1474,24] := 2.0;
   DATA[1474,25] := 2.0;
   DATA[1474,26] := 7.876378;
   DATA[1474,27] := 142.3994;
   DATA[1474,28] := 263.0095;
   DATA[1474,29] := 12.11228;
   DATA[1474,30] := 1.720456;
   DATA[1474,31] := 1.287306;
   DATA[1474,32] := 0.7352687;
   DATA[1474,33] := 0.3106043;
   DATA[1474,34] := 2.0;
   DATA[1474,35] := 249.7917;
   DATA[1474,36] := 1.730048;
   DATA[1474,37] := 188.5414;
   DATA[1474,38] := 0.000128152;
   DATA[1474,39] := 1.0;
   DATA[1475,1] := 814.1022;
   DATA[1475,2] := 1.0;
   DATA[1475,3] := 1.0;
   DATA[1475,4] := 262.5609;
   DATA[1475,5] := 8.464369;
   DATA[1475,6] := 318.4312;
   DATA[1475,8] := 1.0;
   DATA[1475,9] := 1.0;
   DATA[1475,10] := 1.0;
   DATA[1475,11] := 19.74838;
   DATA[1475,12] := 2.216571;
   DATA[1475,13] := 952.4802;
   DATA[1475,14] := 1.0;
   DATA[1475,15] := 2.0;
   DATA[1475,16] := 1.0;
   DATA[1475,17] := 1.0;
   DATA[1475,18] := 1.0;
   DATA[1475,19] := 2.0;
   DATA[1475,20] := 148.808;
   DATA[1475,21] := 153.3709;
   DATA[1475,22] := 1.711723;
   DATA[1475,23] := 785.7216;
   DATA[1475,24] := 2.0;
   DATA[1475,25] := 2.0;
   DATA[1475,26] := 7.876378;
   DATA[1475,27] := 142.3994;
   DATA[1475,28] := 263.0095;
   DATA[1475,29] := 12.11228;
   DATA[1475,30] := 1.720585;
   DATA[1475,31] := 1.287306;
   DATA[1475,32] := 0.7352687;
   DATA[1475,33] := 0.3106043;
   DATA[1475,34] := 2.0;
   DATA[1475,35] := 249.7917;
   DATA[1475,36] := 1.730048;
   DATA[1475,37] := 188.6215;
   DATA[1475,38] := 0.000128152;
   DATA[1475,39] := 1.0;
   DATA[1476,1] := 813.9844;
   DATA[1476,2] := 1.0;
   DATA[1476,3] := 1.0;
   DATA[1476,4] := 262.5609;
   DATA[1476,5] := 8.464369;
   DATA[1476,6] := 318.4312;
   DATA[1476,8] := 1.0;
   DATA[1476,9] := 1.0;
   DATA[1476,10] := 1.0;
   DATA[1476,11] := 19.74838;
   DATA[1476,12] := 2.216571;
   DATA[1476,13] := 952.2799;
   DATA[1476,14] := 1.0;
   DATA[1476,15] := 2.0;
   DATA[1476,16] := 1.0;
   DATA[1476,17] := 1.0;
   DATA[1476,18] := 1.0;
   DATA[1476,19] := 2.0;
   DATA[1476,20] := 148.808;
   DATA[1476,21] := 153.3709;
   DATA[1476,22] := 1.711723;
   DATA[1476,23] := 785.5294;
   DATA[1476,24] := 2.0;
   DATA[1476,25] := 2.0;
   DATA[1476,26] := 7.876378;
   DATA[1476,27] := 142.3994;
   DATA[1476,28] := 263.0095;
   DATA[1476,29] := 12.11228;
   DATA[1476,30] := 1.722123;
   DATA[1476,31] := 1.282311;
   DATA[1476,32] := 0.7352687;
   DATA[1476,33] := 0.3106043;
   DATA[1476,34] := 2.0;
   DATA[1476,35] := 249.7917;
   DATA[1476,36] := 1.730048;
   DATA[1476,37] := 188.6215;
   DATA[1476,38] := 0.000128152;
   DATA[1476,39] := 1.0;
   DATA[1477,1] := 813.9452;
   DATA[1477,2] := 1.0;
   DATA[1477,3] := 1.0;
   DATA[1477,4] := 262.5609;
   DATA[1477,5] := 8.464369;
   DATA[1477,6] := 318.5337;
   DATA[1477,8] := 1.0;
   DATA[1477,9] := 1.0;
   DATA[1477,10] := 1.0;
   DATA[1477,11] := 19.66835;
   DATA[1477,12] := 2.216571;
   DATA[1477,13] := 951.3987;
   DATA[1477,14] := 1.0;
   DATA[1477,15] := 2.0;
   DATA[1477,16] := 1.0;
   DATA[1477,17] := 1.0;
   DATA[1477,18] := 1.0;
   DATA[1477,19] := 2.0;
   DATA[1477,20] := 148.808;
   DATA[1477,21] := 153.3709;
   DATA[1477,22] := 1.711723;
   DATA[1477,23] := 785.6832;
   DATA[1477,24] := 2.0;
   DATA[1477,25] := 2.0;
   DATA[1477,26] := 7.876378;
   DATA[1477,27] := 142.3994;
   DATA[1477,28] := 263.0095;
   DATA[1477,29] := 12.11228;
   DATA[1477,30] := 1.722123;
   DATA[1477,31] := 1.281927;
   DATA[1477,32] := 0.7352687;
   DATA[1477,33] := 0.309003;
   DATA[1477,34] := 2.0;
   DATA[1477,35] := 249.7917;
   DATA[1477,36] := 1.730048;
   DATA[1477,37] := 188.6215;
   DATA[1477,38] := 0.000128152;
   DATA[1477,39] := 1.0;
   DATA[1478,1] := 814.0237;
   DATA[1478,2] := 1.0;
   DATA[1478,3] := 1.0;
   DATA[1478,4] := 262.5609;
   DATA[1478,5] := 8.464369;
   DATA[1478,6] := 318.585;
   DATA[1478,8] := 1.0;
   DATA[1478,9] := 1.0;
   DATA[1478,10] := 1.0;
   DATA[1478,11] := 19.66835;
   DATA[1478,12] := 2.216571;
   DATA[1478,13] := 951.2786;
   DATA[1478,14] := 1.0;
   DATA[1478,15] := 2.0;
   DATA[1478,16] := 1.0;
   DATA[1478,17] := 1.0;
   DATA[1478,18] := 1.0;
   DATA[1478,19] := 2.0;
   DATA[1478,20] := 148.808;
   DATA[1478,21] := 153.3709;
   DATA[1478,22] := 1.711723;
   DATA[1478,23] := 785.837;
   DATA[1478,24] := 2.0;
   DATA[1478,25] := 2.0;
   DATA[1478,26] := 7.876378;
   DATA[1478,27] := 142.3994;
   DATA[1478,28] := 263.0095;
   DATA[1478,29] := 12.11228;
   DATA[1478,30] := 1.722123;
   DATA[1478,31] := 1.288203;
   DATA[1478,32] := 0.7352687;
   DATA[1478,33] := 0.3083624;
   DATA[1478,34] := 2.0;
   DATA[1478,35] := 249.6155;
   DATA[1478,36] := 1.730048;
   DATA[1478,37] := 188.6215;
   DATA[1478,38] := 0.000128152;
   DATA[1478,39] := 1.0;
   DATA[1479,1] := 814.0237;
   DATA[1479,2] := 1.0;
   DATA[1479,3] := 1.0;
   DATA[1479,4] := 262.5609;
   DATA[1479,5] := 8.464369;
   DATA[1479,6] := 318.585;
   DATA[1479,8] := 1.0;
   DATA[1479,9] := 1.0;
   DATA[1479,10] := 1.0;
   DATA[1479,11] := 19.75479;
   DATA[1479,12] := 2.216571;
   DATA[1479,13] := 950.5576;
   DATA[1479,14] := 1.0;
   DATA[1479,15] := 2.0;
   DATA[1479,16] := 1.0;
   DATA[1479,17] := 1.0;
   DATA[1479,18] := 1.0;
   DATA[1479,19] := 2.0;
   DATA[1479,20] := 148.808;
   DATA[1479,21] := 153.3709;
   DATA[1479,22] := 1.710698;
   DATA[1479,23] := 785.9139;
   DATA[1479,24] := 2.0;
   DATA[1479,25] := 2.0;
   DATA[1479,26] := 7.876378;
   DATA[1479,27] := 142.3994;
   DATA[1479,28] := 263.0095;
   DATA[1479,29] := 12.11228;
   DATA[1479,30] := 1.722123;
   DATA[1479,31] := 1.285129;
   DATA[1479,32] := 0.7352687;
   DATA[1479,33] := 0.3102841;
   DATA[1479,34] := 2.0;
   DATA[1479,35] := 249.5995;
   DATA[1479,36] := 1.665972;
   DATA[1479,37] := 188.6215;
   DATA[1479,38] := 0.000128152;
   DATA[1479,39] := 1.0;
   DATA[1480,1] := 814.1807;
   DATA[1480,2] := 1.0;
   DATA[1480,3] := 1.0;
   DATA[1480,4] := 262.5609;
   DATA[1480,5] := 8.464369;
   DATA[1480,6] := 318.585;
   DATA[1480,8] := 1.0;
   DATA[1480,9] := 1.0;
   DATA[1480,10] := 1.0;
   DATA[1480,11] := 19.75799;
   DATA[1480,12] := 2.218108;
   DATA[1480,13] := 950.3973;
   DATA[1480,14] := 1.0;
   DATA[1480,15] := 2.0;
   DATA[1480,16] := 1.0;
   DATA[1480,17] := 1.0;
   DATA[1480,18] := 1.0;
   DATA[1480,19] := 2.0;
   DATA[1480,20] := 148.808;
   DATA[1480,21] := 153.3709;
   DATA[1480,22] := 1.709544;
   DATA[1480,23] := 785.9523;
   DATA[1480,24] := 2.0;
   DATA[1480,25] := 2.0;
   DATA[1480,26] := 7.876378;
   DATA[1480,27] := 142.3994;
   DATA[1480,28] := 263.0095;
   DATA[1480,29] := 12.11228;
   DATA[1480,30] := 1.722123;
   DATA[1480,31] := 1.296913;
   DATA[1480,32] := 0.7352687;
   DATA[1480,33] := 0.3108606;
   DATA[1480,34] := 2.0;
   DATA[1480,35] := 249.5995;
   DATA[1480,36] := 1.665972;
   DATA[1480,37] := 188.6215;
   DATA[1480,38] := 0.000128152;
   DATA[1480,39] := 1.0;
   DATA[1481,1] := 814.22;
   DATA[1481,2] := 1.0;
   DATA[1481,3] := 1.0;
   DATA[1481,4] := 262.5609;
   DATA[1481,5] := 8.464369;
   DATA[1481,6] := 318.585;
   DATA[1481,8] := 1.0;
   DATA[1481,9] := 1.0;
   DATA[1481,10] := 1.0;
   DATA[1481,11] := 19.82201;
   DATA[1481,12] := 2.218108;
   DATA[1481,13] := 949.9568;
   DATA[1481,14] := 1.0;
   DATA[1481,15] := 2.0;
   DATA[1481,16] := 1.0;
   DATA[1481,17] := 1.0;
   DATA[1481,18] := 1.0;
   DATA[1481,19] := 2.0;
   DATA[1481,20] := 148.808;
   DATA[1481,21] := 153.3709;
   DATA[1481,22] := 1.709031;
   DATA[1481,23] := 785.7601;
   DATA[1481,24] := 2.0;
   DATA[1481,25] := 2.0;
   DATA[1481,26] := 7.876378;
   DATA[1481,27] := 142.3994;
   DATA[1481,28] := 263.0095;
   DATA[1481,29] := 12.11228;
   DATA[1481,30] := 1.720585;
   DATA[1481,31] := 1.308697;
   DATA[1481,32] := 0.7352687;
   DATA[1481,33] := 0.3103481;
   DATA[1481,34] := 2.0;
   DATA[1481,35] := 249.5995;
   DATA[1481,36] := 1.665972;
   DATA[1481,37] := 188.4453;
   DATA[1481,38] := 0.000128152;
   DATA[1481,39] := 1.0;
   DATA[1482,1] := 813.8275;
   DATA[1482,2] := 1.0;
   DATA[1482,3] := 1.0;
   DATA[1482,4] := 262.5609;
   DATA[1482,5] := 8.464369;
   DATA[1482,6] := 318.585;
   DATA[1482,8] := 1.0;
   DATA[1482,9] := 1.0;
   DATA[1482,10] := 1.0;
   DATA[1482,11] := 19.82201;
   DATA[1482,12] := 2.217083;
   DATA[1482,13] := 949.3159;
   DATA[1482,14] := 1.0;
   DATA[1482,15] := 2.0;
   DATA[1482,16] := 1.0;
   DATA[1482,17] := 1.0;
   DATA[1482,18] := 1.0;
   DATA[1482,19] := 2.0;
   DATA[1482,20] := 148.808;
   DATA[1482,21] := 153.3709;
   DATA[1482,22] := 1.708775;
   DATA[1482,23] := 786.0292;
   DATA[1482,24] := 2.0;
   DATA[1482,25] := 2.0;
   DATA[1482,26] := 7.876378;
   DATA[1482,27] := 142.3994;
   DATA[1482,28] := 263.0095;
   DATA[1482,29] := 12.11228;
   DATA[1482,30] := 1.719046;
   DATA[1482,31] := 1.304598;
   DATA[1482,32] := 0.7352687;
   DATA[1482,33] := 0.3084265;
   DATA[1482,34] := 2.0;
   DATA[1482,35] := 249.5995;
   DATA[1482,36] := 1.665972;
   DATA[1482,37] := 188.4453;
   DATA[1482,38] := 0.000128152;
   DATA[1482,39] := 1.0;
   DATA[1483,1] := 814.5732;
   DATA[1483,2] := 1.0;
   DATA[1483,3] := 1.0;
   DATA[1483,4] := 262.5609;
   DATA[1483,5] := 8.464369;
   DATA[1483,6] := 318.585;
   DATA[1483,8] := 1.0;
   DATA[1483,9] := 1.0;
   DATA[1483,10] := 1.0;
   DATA[1483,11] := 19.82201;
   DATA[1483,12] := 2.214265;
   DATA[1483,13] := 948.4748;
   DATA[1483,14] := 1.0;
   DATA[1483,15] := 2.0;
   DATA[1483,16] := 1.0;
   DATA[1483,17] := 1.0;
   DATA[1483,18] := 1.0;
   DATA[1483,19] := 2.0;
   DATA[1483,20] := 148.808;
   DATA[1483,21] := 153.3709;
   DATA[1483,22] := 1.706597;
   DATA[1483,23] := 785.7216;
   DATA[1483,24] := 2.0;
   DATA[1483,25] := 2.0;
   DATA[1483,26] := 7.876378;
   DATA[1483,27] := 142.3994;
   DATA[1483,28] := 263.0095;
   DATA[1483,29] := 12.11228;
   DATA[1483,30] := 1.719046;
   DATA[1483,31] := 1.292046;
   DATA[1483,32] := 0.7352687;
   DATA[1483,33] := 0.3084265;
   DATA[1483,34] := 2.0;
   DATA[1483,35] := 249.4392;
   DATA[1483,36] := 1.665972;
   DATA[1483,37] := 188.4453;
   DATA[1483,38] := 0.000128152;
   DATA[1483,39] := 1.0;
   DATA[1484,1] := 814.3377;
   DATA[1484,2] := 1.0;
   DATA[1484,3] := 1.0;
   DATA[1484,4] := 262.5609;
   DATA[1484,5] := 8.464369;
   DATA[1484,6] := 318.585;
   DATA[1484,8] := 1.0;
   DATA[1484,9] := 1.0;
   DATA[1484,10] := 1.0;
   DATA[1484,11] := 19.77399;
   DATA[1484,12] := 2.214265;
   DATA[1484,13] := 948.5148;
   DATA[1484,14] := 1.0;
   DATA[1484,15] := 2.0;
   DATA[1484,16] := 1.0;
   DATA[1484,17] := 1.0;
   DATA[1484,18] := 1.0;
   DATA[1484,19] := 2.0;
   DATA[1484,20] := 148.808;
   DATA[1484,21] := 153.3709;
   DATA[1484,22] := 1.705571;
   DATA[1484,23] := 786.0677;
   DATA[1484,24] := 2.0;
   DATA[1484,25] := 2.0;
   DATA[1484,26] := 7.876378;
   DATA[1484,27] := 142.3994;
   DATA[1484,28] := 263.0095;
   DATA[1484,29] := 12.11228;
   DATA[1484,30] := 1.719046;
   DATA[1484,31] := 1.292046;
   DATA[1484,32] := 0.7352687;
   DATA[1484,33] := 0.3084265;
   DATA[1484,34] := 2.0;
   DATA[1484,35] := 249.4392;
   DATA[1484,36] := 1.665972;
   DATA[1484,37] := 188.4453;
   DATA[1484,38] := 0.000128152;
   DATA[1484,39] := 1.0;
   DATA[1485,1] := 814.4948;
   DATA[1485,2] := 1.0;
   DATA[1485,3] := 1.0;
   DATA[1485,4] := 262.5609;
   DATA[1485,5] := 8.464369;
   DATA[1485,6] := 318.585;
   DATA[1485,8] := 1.0;
   DATA[1485,9] := 1.0;
   DATA[1485,10] := 1.0;
   DATA[1485,11] := 19.75799;
   DATA[1485,12] := 2.214649;
   DATA[1485,13] := 947.874;
   DATA[1485,14] := 1.0;
   DATA[1485,15] := 2.0;
   DATA[1485,16] := 1.0;
   DATA[1485,17] := 1.0;
   DATA[1485,18] := 1.0;
   DATA[1485,19] := 2.0;
   DATA[1485,20] := 148.808;
   DATA[1485,21] := 153.3709;
   DATA[1485,22] := 1.707622;
   DATA[1485,23] := 786.2984;
   DATA[1485,24] := 2.0;
   DATA[1485,25] := 2.0;
   DATA[1485,26] := 7.876378;
   DATA[1485,27] := 142.3994;
   DATA[1485,28] := 263.0095;
   DATA[1485,29] := 12.11228;
   DATA[1485,30] := 1.719046;
   DATA[1485,31] := 1.292046;
   DATA[1485,32] := 0.7352687;
   DATA[1485,33] := 0.3084265;
   DATA[1485,34] := 2.0;
   DATA[1485,35] := 249.4553;
   DATA[1485,36] := 1.665972;
   DATA[1485,37] := 188.4453;
   DATA[1485,38] := 0.000128152;
   DATA[1485,39] := 1.0;
   DATA[1486,1] := 814.6125;
   DATA[1486,2] := 1.0;
   DATA[1486,3] := 1.0;
   DATA[1486,4] := 262.5609;
   DATA[1486,5] := 8.464369;
   DATA[1486,6] := 318.585;
   DATA[1486,8] := 1.0;
   DATA[1486,9] := 1.0;
   DATA[1486,10] := 1.0;
   DATA[1486,11] := 19.73558;
   DATA[1486,12] := 2.214649;
   DATA[1486,13] := 947.4734;
   DATA[1486,14] := 1.0;
   DATA[1486,15] := 2.0;
   DATA[1486,16] := 1.0;
   DATA[1486,17] := 1.0;
   DATA[1486,18] := 1.0;
   DATA[1486,19] := 2.0;
   DATA[1486,20] := 148.808;
   DATA[1486,21] := 153.3709;
   DATA[1486,22] := 1.708775;
   DATA[1486,23] := 786.2215;
   DATA[1486,24] := 2.0;
   DATA[1486,25] := 2.0;
   DATA[1486,26] := 7.876378;
   DATA[1486,27] := 142.3994;
   DATA[1486,28] := 263.0095;
   DATA[1486,29] := 12.11228;
   DATA[1486,30] := 1.719046;
   DATA[1486,31] := 1.297041;
   DATA[1486,32] := 0.7352687;
   DATA[1486,33] := 0.3084265;
   DATA[1486,34] := 2.0;
   DATA[1486,35] := 249.7917;
   DATA[1486,36] := 1.665972;
   DATA[1486,37] := 188.6055;
   DATA[1486,38] := 0.000128152;
   DATA[1486,39] := 1.0;
   DATA[1487,1] := 815.005;
   DATA[1487,2] := 1.0;
   DATA[1487,3] := 1.0;
   DATA[1487,4] := 262.5609;
   DATA[1487,5] := 8.464369;
   DATA[1487,6] := 318.585;
   DATA[1487,8] := 1.0;
   DATA[1487,9] := 1.0;
   DATA[1487,10] := 1.0;
   DATA[1487,11] := 19.73558;
   DATA[1487,12] := 2.214649;
   DATA[1487,13] := 947.3132;
   DATA[1487,14] := 1.0;
   DATA[1487,15] := 2.0;
   DATA[1487,16] := 1.0;
   DATA[1487,17] := 1.0;
   DATA[1487,18] := 1.0;
   DATA[1487,19] := 2.0;
   DATA[1487,20] := 148.808;
   DATA[1487,21] := 153.3709;
   DATA[1487,22] := 1.710313;
   DATA[1487,23] := 786.1061;
   DATA[1487,24] := 2.0;
   DATA[1487,25] := 2.0;
   DATA[1487,26] := 7.876378;
   DATA[1487,27] := 142.3994;
   DATA[1487,28] := 263.0095;
   DATA[1487,29] := 12.11228;
   DATA[1487,30] := 1.719687;
   DATA[1487,31] := 1.30114;
   DATA[1487,32] := 0.7352687;
   DATA[1487,33] := 0.3084265;
   DATA[1487,34] := 2.0;
   DATA[1487,35] := 249.7917;
   DATA[1487,36] := 1.665972;
   DATA[1487,37] := 188.7016;
   DATA[1487,38] := 0.000128152;
   DATA[1487,39] := 1.0;
   DATA[1488,1] := 815.3975;
   DATA[1488,2] := 1.0;
   DATA[1488,3] := 1.0;
   DATA[1488,4] := 262.5609;
   DATA[1488,5] := 8.464369;
   DATA[1488,6] := 318.585;
   DATA[1488,8] := 1.0;
   DATA[1488,9] := 1.0;
   DATA[1488,10] := 1.0;
   DATA[1488,11] := 19.81241;
   DATA[1488,12] := 2.214649;
   DATA[1488,13] := 947.2731;
   DATA[1488,14] := 1.0;
   DATA[1488,15] := 2.0;
   DATA[1488,16] := 1.0;
   DATA[1488,17] := 1.0;
   DATA[1488,18] := 1.0;
   DATA[1488,19] := 2.0;
   DATA[1488,20] := 148.808;
   DATA[1488,21] := 153.3709;
   DATA[1488,22] := 1.711466;
   DATA[1488,23] := 786.4522;
   DATA[1488,24] := 2.0;
   DATA[1488,25] := 2.0;
   DATA[1488,26] := 7.876378;
   DATA[1488,27] := 142.3994;
   DATA[1488,28] := 263.0095;
   DATA[1488,29] := 12.11228;
   DATA[1488,30] := 1.72161;
   DATA[1488,31] := 1.298578;
   DATA[1488,32] := 0.7352687;
   DATA[1488,33] := 0.3084265;
   DATA[1488,34] := 2.0;
   DATA[1488,35] := 249.7917;
   DATA[1488,36] := 1.665972;
   DATA[1488,37] := 188.7016;
   DATA[1488,38] := 0.000128152;
   DATA[1488,39] := 1.0;
   DATA[1489,1] := 815.5153;
   DATA[1489,2] := 1.0;
   DATA[1489,3] := 1.0;
   DATA[1489,4] := 262.5609;
   DATA[1489,5] := 8.464369;
   DATA[1489,6] := 318.585;
   DATA[1489,8] := 1.0;
   DATA[1489,9] := 1.0;
   DATA[1489,10] := 1.0;
   DATA[1489,11] := 19.83162;
   DATA[1489,12] := 2.214649;
   DATA[1489,13] := 946.7925;
   DATA[1489,14] := 1.0;
   DATA[1489,15] := 2.0;
   DATA[1489,16] := 1.0;
   DATA[1489,17] := 1.0;
   DATA[1489,18] := 1.0;
   DATA[1489,19] := 2.0;
   DATA[1489,20] := 148.808;
   DATA[1489,21] := 153.3709;
   DATA[1489,22] := 1.71262;
   DATA[1489,23] := 786.2984;
   DATA[1489,24] := 2.0;
   DATA[1489,25] := 2.0;
   DATA[1489,26] := 7.876378;
   DATA[1489,27] := 142.3994;
   DATA[1489,28] := 263.0095;
   DATA[1489,29] := 12.11228;
   DATA[1489,30] := 1.721866;
   DATA[1489,31] := 1.299475;
   DATA[1489,32] := 0.7352687;
   DATA[1489,33] := 0.3084265;
   DATA[1489,34] := 2.0;
   DATA[1489,35] := 249.7917;
   DATA[1489,36] := 1.665972;
   DATA[1489,37] := 188.7016;
   DATA[1489,38] := 0.000128152;
   DATA[1489,39] := 1.0;
   DATA[1490,1] := 815.3583;
   DATA[1490,2] := 1.0;
   DATA[1490,3] := 1.0;
   DATA[1490,4] := 262.5609;
   DATA[1490,5] := 8.464369;
   DATA[1490,6] := 318.585;
   DATA[1490,8] := 1.0;
   DATA[1490,9] := 1.0;
   DATA[1490,10] := 1.0;
   DATA[1490,11] := 19.84762;
   DATA[1490,12] := 2.214649;
   DATA[1490,13] := 946.3519;
   DATA[1490,14] := 1.0;
   DATA[1490,15] := 2.0;
   DATA[1490,16] := 1.0;
   DATA[1490,17] := 1.0;
   DATA[1490,18] := 1.0;
   DATA[1490,19] := 2.0;
   DATA[1490,20] := 148.808;
   DATA[1490,21] := 153.3709;
   DATA[1490,22] := 1.712748;
   DATA[1490,23] := 786.4907;
   DATA[1490,24] := 2.0;
   DATA[1490,25] := 2.0;
   DATA[1490,26] := 7.876378;
   DATA[1490,27] := 142.3994;
   DATA[1490,28] := 263.0095;
   DATA[1490,29] := 12.11228;
   DATA[1490,30] := 1.721866;
   DATA[1490,31] := 1.300115;
   DATA[1490,32] := 0.7352687;
   DATA[1490,33] := 0.3084265;
   DATA[1490,34] := 2.0;
   DATA[1490,35] := 249.7917;
   DATA[1490,36] := 1.665972;
   DATA[1490,37] := 188.7016;
   DATA[1490,38] := 0.000128152;
   DATA[1490,39] := 1.0;
   DATA[1491,1] := 815.9471;
   DATA[1491,2] := 1.0;
   DATA[1491,3] := 1.0;
   DATA[1491,4] := 262.5609;
   DATA[1491,5] := 8.464369;
   DATA[1491,6] := 318.585;
   DATA[1491,8] := 1.0;
   DATA[1491,9] := 1.0;
   DATA[1491,10] := 1.0;
   DATA[1491,11] := 19.84762;
   DATA[1491,12] := 2.214137;
   DATA[1491,13] := 945.8713;
   DATA[1491,14] := 1.0;
   DATA[1491,15] := 2.0;
   DATA[1491,16] := 1.0;
   DATA[1491,17] := 1.0;
   DATA[1491,18] := 1.0;
   DATA[1491,19] := 2.0;
   DATA[1491,20] := 148.808;
   DATA[1491,21] := 153.3709;
   DATA[1491,22] := 1.712748;
   DATA[1491,23] := 786.5291;
   DATA[1491,24] := 2.0;
   DATA[1491,25] := 2.0;
   DATA[1491,26] := 7.876378;
   DATA[1491,27] := 142.3994;
   DATA[1491,28] := 263.0095;
   DATA[1491,29] := 12.11228;
   DATA[1491,30] := 1.724045;
   DATA[1491,31] := 1.284104;
   DATA[1491,32] := 0.7352687;
   DATA[1491,33] := 0.3084265;
   DATA[1491,34] := 2.0;
   DATA[1491,35] := 250.0;
   DATA[1491,36] := 1.665972;
   DATA[1491,37] := 188.7016;
   DATA[1491,38] := 0.000128152;
   DATA[1491,39] := 1.0;
   DATA[1492,1] := 815.5938;
   DATA[1492,2] := 1.0;
   DATA[1492,3] := 1.0;
   DATA[1492,4] := 262.5609;
   DATA[1492,5] := 8.464369;
   DATA[1492,6] := 318.585;
   DATA[1492,8] := 1.0;
   DATA[1492,9] := 1.0;
   DATA[1492,10] := 1.0;
   DATA[1492,11] := 19.81241;
   DATA[1492,12] := 2.213881;
   DATA[1492,13] := 945.5909;
   DATA[1492,14] := 1.0;
   DATA[1492,15] := 2.0;
   DATA[1492,16] := 1.0;
   DATA[1492,17] := 1.0;
   DATA[1492,18] := 1.0;
   DATA[1492,19] := 2.0;
   DATA[1492,20] := 148.808;
   DATA[1492,21] := 153.3709;
   DATA[1492,22] := 1.712748;
   DATA[1492,23] := 786.8752;
   DATA[1492,24] := 2.0;
   DATA[1492,25] := 2.0;
   DATA[1492,26] := 7.876378;
   DATA[1492,27] := 142.3994;
   DATA[1492,28] := 263.0095;
   DATA[1492,29] := 12.11228;
   DATA[1492,30] := 1.724173;
   DATA[1492,31] := 1.28641;
   DATA[1492,32] := 0.7352687;
   DATA[1492,33] := 0.3084265;
   DATA[1492,34] := 2.0;
   DATA[1492,35] := 250.0961;
   DATA[1492,36] := 1.665972;
   DATA[1492,37] := 188.7657;
   DATA[1492,38] := 0.000128152;
   DATA[1492,39] := 1.0;
   DATA[1493,1] := 815.8686;
   DATA[1493,2] := 1.0;
   DATA[1493,3] := 1.0;
   DATA[1493,4] := 262.5609;
   DATA[1493,5] := 8.464369;
   DATA[1493,6] := 318.585;
   DATA[1493,8] := 1.0;
   DATA[1493,9] := 1.0;
   DATA[1493,10] := 1.0;
   DATA[1493,11] := 19.81241;
   DATA[1493,12] := 2.213881;
   DATA[1493,13] := 945.3105;
   DATA[1493,14] := 1.0;
   DATA[1493,15] := 2.0;
   DATA[1493,16] := 1.0;
   DATA[1493,17] := 1.0;
   DATA[1493,18] := 1.0;
   DATA[1493,19] := 2.0;
   DATA[1493,20] := 148.808;
   DATA[1493,21] := 153.3709;
   DATA[1493,22] := 1.712748;
   DATA[1493,23] := 786.9905;
   DATA[1493,24] := 2.0;
   DATA[1493,25] := 2.0;
   DATA[1493,26] := 7.876378;
   DATA[1493,27] := 142.3994;
   DATA[1493,28] := 263.0095;
   DATA[1493,29] := 12.11228;
   DATA[1493,30] := 1.724173;
   DATA[1493,31] := 1.282567;
   DATA[1493,32] := 0.7352687;
   DATA[1493,33] := 0.3084265;
   DATA[1493,34] := 2.0;
   DATA[1493,35] := 250.0961;
   DATA[1493,36] := 1.665972;
   DATA[1493,37] := 188.7657;
   DATA[1493,38] := 0.000128152;
   DATA[1493,39] := 1.0;
   DATA[1494,1] := 815.8686;
   DATA[1494,2] := 1.0;
   DATA[1494,3] := 1.0;
   DATA[1494,4] := 262.5609;
   DATA[1494,5] := 8.464369;
   DATA[1494,6] := 318.6363;
   DATA[1494,8] := 1.0;
   DATA[1494,9] := 1.0;
   DATA[1494,10] := 1.0;
   DATA[1494,11] := 19.81241;
   DATA[1494,12] := 2.213881;
   DATA[1494,13] := 944.5895;
   DATA[1494,14] := 1.0;
   DATA[1494,15] := 2.0;
   DATA[1494,16] := 1.0;
   DATA[1494,17] := 1.0;
   DATA[1494,18] := 1.0;
   DATA[1494,19] := 2.0;
   DATA[1494,20] := 148.808;
   DATA[1494,21] := 153.3709;
   DATA[1494,22] := 1.712748;
   DATA[1494,23] := 787.4904;
   DATA[1494,24] := 2.0;
   DATA[1494,25] := 2.0;
   DATA[1494,26] := 7.876378;
   DATA[1494,27] := 142.3994;
   DATA[1494,28] := 263.0095;
   DATA[1494,29] := 12.11228;
   DATA[1494,30] := 1.724173;
   DATA[1494,31] := 1.284104;
   DATA[1494,32] := 0.7352687;
   DATA[1494,33] := 0.3084265;
   DATA[1494,34] := 2.0;
   DATA[1494,35] := 249.7917;
   DATA[1494,36] := 1.665972;
   DATA[1494,37] := 188.7657;
   DATA[1494,38] := 0.000128152;
   DATA[1494,39] := 1.0;
   DATA[1495,1] := 815.5938;
   DATA[1495,2] := 1.0;
   DATA[1495,3] := 1.0;
   DATA[1495,4] := 262.5609;
   DATA[1495,5] := 8.464369;
   DATA[1495,6] := 318.6363;
   DATA[1495,8] := 1.0;
   DATA[1495,9] := 1.0;
   DATA[1495,10] := 1.0;
   DATA[1495,11] := 19.81241;
   DATA[1495,12] := 2.213881;
   DATA[1495,13] := 944.4694;
   DATA[1495,14] := 1.0;
   DATA[1495,15] := 2.0;
   DATA[1495,16] := 1.0;
   DATA[1495,17] := 1.0;
   DATA[1495,18] := 1.0;
   DATA[1495,19] := 2.0;
   DATA[1495,20] := 148.808;
   DATA[1495,21] := 153.3709;
   DATA[1495,22] := 1.710698;
   DATA[1495,23] := 787.7595;
   DATA[1495,24] := 2.0;
   DATA[1495,25] := 2.0;
   DATA[1495,26] := 7.876378;
   DATA[1495,27] := 142.4507;
   DATA[1495,28] := 263.2658;
   DATA[1495,29] := 12.11228;
   DATA[1495,30] := 1.724173;
   DATA[1495,31] := 1.292558;
   DATA[1495,32] := 0.7352687;
   DATA[1495,33] := 0.3084265;
   DATA[1495,34] := 2.0;
   DATA[1495,35] := 249.7917;
   DATA[1495,36] := 1.665972;
   DATA[1495,37] := 188.7657;
   DATA[1495,38] := 0.000128152;
   DATA[1495,39] := 1.0;
   DATA[1496,1] := 815.8686;
   DATA[1496,2] := 1.0;
   DATA[1496,3] := 1.0;
   DATA[1496,4] := 262.5609;
   DATA[1496,5] := 8.464369;
   DATA[1496,6] := 318.6363;
   DATA[1496,8] := 1.0;
   DATA[1496,9] := 1.0;
   DATA[1496,10] := 1.0;
   DATA[1496,11] := 19.87963;
   DATA[1496,12] := 2.212728;
   DATA[1496,13] := 943.9487;
   DATA[1496,14] := 1.0;
   DATA[1496,15] := 2.0;
   DATA[1496,16] := 1.0;
   DATA[1496,17] := 1.0;
   DATA[1496,18] := 1.0;
   DATA[1496,19] := 2.0;
   DATA[1496,20] := 148.808;
   DATA[1496,21] := 153.3709;
   DATA[1496,22] := 1.713389;
   DATA[1496,23] := 787.7595;
   DATA[1496,24] := 2.0;
   DATA[1496,25] := 2.0;
   DATA[1496,26] := 7.876378;
   DATA[1496,27] := 142.5276;
   DATA[1496,28] := 263.2658;
   DATA[1496,29] := 12.11228;
   DATA[1496,30] := 1.724173;
   DATA[1496,31] := 1.286666;
   DATA[1496,32] := 0.7352687;
   DATA[1496,33] := 0.3098997;
   DATA[1496,34] := 2.0;
   DATA[1496,35] := 249.7917;
   DATA[1496,36] := 1.665972;
   DATA[1496,37] := 188.7657;
   DATA[1496,38] := 0.000128152;
   DATA[1496,39] := 1.0;
   DATA[1497,1] := 815.5546;
   DATA[1497,2] := 1.0;
   DATA[1497,3] := 1.0;
   DATA[1497,4] := 262.5609;
   DATA[1497,5] := 8.464369;
   DATA[1497,6] := 318.6363;
   DATA[1497,8] := 1.0;
   DATA[1497,9] := 1.0;
   DATA[1497,10] := 1.0;
   DATA[1497,11] := 19.87963;
   DATA[1497,12] := 2.212728;
   DATA[1497,13] := 943.3879;
   DATA[1497,14] := 1.0;
   DATA[1497,15] := 2.0;
   DATA[1497,16] := 1.0;
   DATA[1497,17] := 1.0;
   DATA[1497,18] := 1.0;
   DATA[1497,19] := 2.0;
   DATA[1497,20] := 148.808;
   DATA[1497,21] := 153.3709;
   DATA[1497,22] := 1.713389;
   DATA[1497,23] := 788.0671;
   DATA[1497,24] := 2.0;
   DATA[1497,25] := 2.0;
   DATA[1497,26] := 7.876378;
   DATA[1497,27] := 142.5276;
   DATA[1497,28] := 263.2658;
   DATA[1497,29] := 12.11228;
   DATA[1497,30] := 1.724173;
   DATA[1497,31] := 1.28167;
   DATA[1497,32] := 0.7352687;
   DATA[1497,33] := 0.3098997;
   DATA[1497,34] := 2.0;
   DATA[1497,35] := 249.7917;
   DATA[1497,36] := 1.665972;
   DATA[1497,37] := 188.7977;
   DATA[1497,38] := 0.000128152;
   DATA[1497,39] := 1.0;
   DATA[1498,1] := 815.5153;
   DATA[1498,2] := 1.0;
   DATA[1498,3] := 1.0;
   DATA[1498,4] := 262.5609;
   DATA[1498,5] := 8.464369;
   DATA[1498,6] := 318.6363;
   DATA[1498,8] := 1.0;
   DATA[1498,9] := 1.0;
   DATA[1498,10] := 1.0;
   DATA[1498,11] := 19.91165;
   DATA[1498,12] := 2.212728;
   DATA[1498,13] := 942.667;
   DATA[1498,14] := 1.0;
   DATA[1498,15] := 2.0;
   DATA[1498,16] := 1.0;
   DATA[1498,17] := 1.0;
   DATA[1498,18] := 1.0;
   DATA[1498,19] := 2.0;
   DATA[1498,20] := 148.808;
   DATA[1498,21] := 153.5504;
   DATA[1498,22] := 1.711595;
   DATA[1498,23] := 788.4132;
   DATA[1498,24] := 2.0;
   DATA[1498,25] := 2.0;
   DATA[1498,26] := 7.876378;
   DATA[1498,27] := 142.5276;
   DATA[1498,28] := 263.2658;
   DATA[1498,29] := 12.11228;
   DATA[1498,30] := 1.724173;
   DATA[1498,31] := 1.263866;
   DATA[1498,32] := 0.7352687;
   DATA[1498,33] := 0.3083624;
   DATA[1498,34] := 2.0;
   DATA[1498,35] := 250.0801;
   DATA[1498,36] := 1.665972;
   DATA[1498,37] := 188.8618;
   DATA[1498,38] := 0.000128152;
   DATA[1498,39] := 1.0;
   DATA[1499,1] := 815.7508;
   DATA[1499,2] := 1.0;
   DATA[1499,3] := 1.0;
   DATA[1499,4] := 262.5609;
   DATA[1499,5] := 8.464369;
   DATA[1499,6] := 318.6363;
   DATA[1499,8] := 1.0;
   DATA[1499,9] := 1.0;
   DATA[1499,10] := 1.0;
   DATA[1499,11] := 19.91165;
   DATA[1499,12] := 2.212728;
   DATA[1499,13] := 942.1462;
   DATA[1499,14] := 1.0;
   DATA[1499,15] := 2.0;
   DATA[1499,16] := 1.0;
   DATA[1499,17] := 1.0;
   DATA[1499,18] := 1.0;
   DATA[1499,19] := 2.0;
   DATA[1499,20] := 148.808;
   DATA[1499,21] := 153.5504;
   DATA[1499,22] := 1.711338;
   DATA[1499,23] := 788.6439;
   DATA[1499,24] := 2.0;
   DATA[1499,25] := 2.0;
   DATA[1499,26] := 7.876378;
   DATA[1499,27] := 142.5276;
   DATA[1499,28] := 263.2658;
   DATA[1499,29] := 12.11228;
   DATA[1499,30] := 1.722379;
   DATA[1499,31] := 1.270398;
   DATA[1499,32] := 0.7352687;
   DATA[1499,33] := 0.3083624;
   DATA[1499,34] := 2.0;
   DATA[1499,35] := 250.1602;
   DATA[1499,36] := 1.665972;
   DATA[1499,37] := 189.006;
   DATA[1499,38] := 0.000128152;
   DATA[1499,39] := 1.0;
   DATA[1500,1] := 815.7901;
   DATA[1500,2] := 1.0;
   DATA[1500,3] := 1.0;
   DATA[1500,4] := 262.5609;
   DATA[1500,5] := 8.464369;
   DATA[1500,6] := 318.6363;
   DATA[1500,8] := 1.0;
   DATA[1500,9] := 1.0;
   DATA[1500,10] := 1.0;
   DATA[1500,11] := 19.85082;
   DATA[1500,12] := 2.212728;
   DATA[1500,13] := 941.5054;
   DATA[1500,14] := 1.0;
   DATA[1500,15] := 2.0;
   DATA[1500,16] := 1.0;
   DATA[1500,17] := 1.0;
   DATA[1500,18] := 1.0;
   DATA[1500,19] := 2.0;
   DATA[1500,20] := 148.808;
   DATA[1500,21] := 153.5504;
   DATA[1500,22] := 1.711338;
   DATA[1500,23] := 789.0284;
   DATA[1500,24] := 2.0;
   DATA[1500,25] := 2.0;
   DATA[1500,26] := 7.876378;
   DATA[1500,27] := 142.5276;
   DATA[1500,28] := 263.1377;
   DATA[1500,29] := 12.11228;
   DATA[1500,30] := 1.721738;
   DATA[1500,31] := 1.291277;
   DATA[1500,32] := 0.7352687;
   DATA[1500,33] := 0.3093233;
   DATA[1500,34] := 2.0;
   DATA[1500,35] := 250.1602;
   DATA[1500,36] := 1.665972;
   DATA[1500,37] := 189.006;
   DATA[1500,38] := 0.000128152;
   DATA[1500,39] := 1.0;
   DATA[1501,1] := 815.9863;
   DATA[1501,2] := 1.0;
   DATA[1501,3] := 1.0;
   DATA[1501,4] := 262.5609;
   DATA[1501,5] := 8.464369;
   DATA[1501,6] := 318.6363;
   DATA[1501,8] := 1.0;
   DATA[1501,9] := 1.0;
   DATA[1501,10] := 1.0;
   DATA[1501,11] := 19.82201;
   DATA[1501,12] := 2.212728;
   DATA[1501,13] := 941.0648;
   DATA[1501,14] := 1.0;
   DATA[1501,15] := 2.0;
   DATA[1501,16] := 1.0;
   DATA[1501,17] := 1.0;
   DATA[1501,18] := 1.0;
   DATA[1501,19] := 2.0;
   DATA[1501,20] := 148.808;
   DATA[1501,21] := 153.5504;
   DATA[1501,22] := 1.711723;
   DATA[1501,23] := 789.1823;
   DATA[1501,24] := 2.0;
   DATA[1501,25] := 2.0;
   DATA[1501,26] := 7.876378;
   DATA[1501,27] := 142.5276;
   DATA[1501,28] := 263.1377;
   DATA[1501,29] := 12.11228;
   DATA[1501,30] := 1.721738;
   DATA[1501,31] := 1.29307;
   DATA[1501,32] := 0.7352687;
   DATA[1501,33] := 0.3093233;
   DATA[1501,34] := 2.0;
   DATA[1501,35] := 250.1602;
   DATA[1501,36] := 1.665972;
   DATA[1501,37] := 189.1342;
   DATA[1501,38] := 0.000128152;
   DATA[1501,39] := 1.0;
   DATA[1502,1] := 815.6723;
   DATA[1502,2] := 1.0;
   DATA[1502,3] := 1.0;
   DATA[1502,4] := 262.5609;
   DATA[1502,5] := 8.464369;
   DATA[1502,6] := 318.6363;
   DATA[1502,8] := 1.0;
   DATA[1502,9] := 1.0;
   DATA[1502,10] := 1.0;
   DATA[1502,11] := 19.7836;
   DATA[1502,12] := 2.212728;
   DATA[1502,13] := 940.6642;
   DATA[1502,14] := 1.0;
   DATA[1502,15] := 2.0;
   DATA[1502,16] := 1.0;
   DATA[1502,17] := 1.0;
   DATA[1502,18] := 1.0;
   DATA[1502,19] := 2.0;
   DATA[1502,20] := 148.808;
   DATA[1502,21] := 153.5504;
   DATA[1502,22] := 1.713004;
   DATA[1502,23] := 789.0284;
   DATA[1502,24] := 2.0;
   DATA[1502,25] := 2.0;
   DATA[1502,26] := 7.876378;
   DATA[1502,27] := 142.5276;
   DATA[1502,28] := 263.1377;
   DATA[1502,29] := 12.11228;
   DATA[1502,30] := 1.721738;
   DATA[1502,31] := 1.308569;
   DATA[1502,32] := 0.7352687;
   DATA[1502,33] := 0.30785;
   DATA[1502,34] := 2.0;
   DATA[1502,35] := 250.1602;
   DATA[1502,36] := 1.665972;
   DATA[1502,37] := 189.1342;
   DATA[1502,38] := 0.000128152;
   DATA[1502,39] := 1.0;
   DATA[1503,1] := 815.6723;
   DATA[1503,2] := 1.0;
   DATA[1503,3] := 1.0;
   DATA[1503,4] := 262.5609;
   DATA[1503,5] := 8.464369;
   DATA[1503,6] := 318.6363;
   DATA[1503,8] := 1.0;
   DATA[1503,9] := 1.0;
   DATA[1503,10] := 1.0;
   DATA[1503,11] := 19.7836;
   DATA[1503,12] := 2.212728;
   DATA[1503,13] := 940.6642;
   DATA[1503,14] := 1.0;
   DATA[1503,15] := 2.0;
   DATA[1503,16] := 1.0;
   DATA[1503,17] := 1.0;
   DATA[1503,18] := 1.0;
   DATA[1503,19] := 2.0;
   DATA[1503,20] := 148.808;
   DATA[1503,21] := 153.5504;
   DATA[1503,22] := 1.713004;
   DATA[1503,23] := 789.0284;
   DATA[1503,24] := 2.0;
   DATA[1503,25] := 2.0;
   DATA[1503,26] := 7.876378;
   DATA[1503,27] := 142.5276;
   DATA[1503,28] := 263.1377;
   DATA[1503,29] := 12.11228;
   DATA[1503,30] := 1.721738;
   DATA[1503,31] := 1.308569;
   DATA[1503,32] := 0.7352687;
   DATA[1503,33] := 0.30785;
   DATA[1503,34] := 2.0;
   DATA[1503,35] := 250.1602;
   DATA[1503,36] := 1.665972;
   DATA[1503,37] := 189.1342;
   DATA[1503,38] := 0.000128152;
   DATA[1503,39] := 1.0;
   DATA[1504,1] := 815.5546;
   DATA[1504,2] := 1.0;
   DATA[1504,3] := 1.0;
   DATA[1504,4] := 262.5609;
   DATA[1504,5] := 8.464369;
   DATA[1504,6] := 318.6363;
   DATA[1504,8] := 1.0;
   DATA[1504,9] := 1.0;
   DATA[1504,10] := 1.0;
   DATA[1504,11] := 19.77079;
   DATA[1504,12] := 2.212728;
   DATA[1504,13] := 940.3439;
   DATA[1504,14] := 1.0;
   DATA[1504,15] := 2.0;
   DATA[1504,16] := 1.0;
   DATA[1504,17] := 1.0;
   DATA[1504,18] := 1.0;
   DATA[1504,19] := 2.0;
   DATA[1504,20] := 148.808;
   DATA[1504,21] := 153.5504;
   DATA[1504,22] := 1.713004;
   DATA[1504,23] := 789.4899;
   DATA[1504,24] := 2.0;
   DATA[1504,25] := 2.0;
   DATA[1504,26] := 7.876378;
   DATA[1504,27] := 142.5276;
   DATA[1504,28] := 263.1377;
   DATA[1504,29] := 12.11228;
   DATA[1504,30] := 1.721738;
   DATA[1504,31] := 1.301524;
   DATA[1504,32] := 0.7352687;
   DATA[1504,33] := 0.30785;
   DATA[1504,34] := 2.0;
   DATA[1504,35] := 250.1602;
   DATA[1504,36] := 1.665972;
   DATA[1504,37] := 189.1342;
   DATA[1504,38] := 0.000128152;
   DATA[1504,39] := 1.0;
   DATA[1505,1] := 815.6723;
   DATA[1505,2] := 1.0;
   DATA[1505,3] := 1.0;
   DATA[1505,4] := 262.5609;
   DATA[1505,5] := 8.464369;
   DATA[1505,6] := 318.9182;
   DATA[1505,8] := 1.0;
   DATA[1505,9] := 1.0;
   DATA[1505,10] := 1.0;
   DATA[1505,11] := 19.77079;
   DATA[1505,12] := 2.210806;
   DATA[1505,13] := 940.1035;
   DATA[1505,14] := 1.0;
   DATA[1505,15] := 2.0;
   DATA[1505,16] := 1.0;
   DATA[1505,17] := 1.0;
   DATA[1505,18] := 1.0;
   DATA[1505,19] := 2.0;
   DATA[1505,20] := 148.808;
   DATA[1505,21] := 153.5504;
   DATA[1505,22] := 1.71262;
   DATA[1505,23] := 789.413;
   DATA[1505,24] := 2.0;
   DATA[1505,25] := 2.0;
   DATA[1505,26] := 7.876378;
   DATA[1505,27] := 142.6814;
   DATA[1505,28] := 263.1377;
   DATA[1505,29] := 12.11228;
   DATA[1505,30] := 1.723148;
   DATA[1505,31] := 1.292814;
   DATA[1505,32] := 0.7352687;
   DATA[1505,33] := 0.3103481;
   DATA[1505,34] := 2.0;
   DATA[1505,35] := 250.1602;
   DATA[1505,36] := 1.665972;
   DATA[1505,37] := 188.7657;
   DATA[1505,38] := 0.000128152;
   DATA[1505,39] := 1.0;
   DATA[1506,1] := 815.2798;
   DATA[1506,2] := 1.0;
   DATA[1506,3] := 1.0;
   DATA[1506,4] := 262.5609;
   DATA[1506,5] := 8.464369;
   DATA[1506,6] := 318.9438;
   DATA[1506,8] := 1.0;
   DATA[1506,9] := 1.0;
   DATA[1506,10] := 1.0;
   DATA[1506,11] := 19.77079;
   DATA[1506,12] := 2.210294;
   DATA[1506,13] := 939.9833;
   DATA[1506,14] := 1.0;
   DATA[1506,15] := 2.0;
